IPC(IP:= DWORD#0, PORT:= WORD#0 , TIME_OUT:= timeout1, IP_C:= IP_C, S_BUF:= COM.S_BUF, R_BUF:= COM.R_BUF, TLS_CONFIG_IN := COM.TLS_CONFIG, useTls:= COM.TLS); (* MQTT Steuerkanal *)

TON_WAIT(IN:=step = last_step AND step > 0,PT:=timeout2);
last_step := step;


(* revision history


*)

END_FUNCTION_BLOCK

// MQTT/Function/InsertStringToBufferAndLength
//returnds new pos in buff
FUNCTION InsertStringToBufferAndLength : UINT
VAR_INPUT
	Str:POINTER TO STRING;
	//address to buffer
	buff:POINTER TO BYTE;
	//Start to insert
	pos:UINT;
	//size of buffer
	//size:UINT;
END_VAR
VAR
	length:UINT;
END_VAR

length := CommonTypesAndFunctions.LEN(Str);
buff[pos]:= OSCAT_BASIC.BYTE_OF_DWORD(in:= length, N:= 1);
buff[pos+1]:= OSCAT_BASIC.BYTE_OF_DWORD(in:= length, N:= 0);

MEM.MemMove(pSource:= str, pDestination:= ADR(buff[pos+2]), uiNumberOfBytes:= length);
InsertStringToBufferAndLength := pos + length + 2;

END_FUNCTION

// MQTT/Function/DoRemainingLength
FUNCTION DoRemainingLength : USINT
VAR_INPUT
	buffer:POINTER TO BYTE;
	RemainingLength:UINT;
	
END_VAR
VAR
	LocalLength:LINT;
	LocalBuffer:ARRAY[0..3]OF BYTE;
	BufferIndex:UINT := 0;
	TmpByte:BYTE;
END_VAR

//check if we have to move data for inserting remaining length
//borders are given in the mqtt doku
//
IF RemainingLength <= 128 THEN
	buffer[1] := UINT_TO_BYTE(RemainingLength);
	DoRemainingLength := 0;
ELSE
	LocalLength := RemainingLength;
	REPEAT
		TmpByte := LINT_TO_BYTE(LocalLength MOD 128);
		LocalLength := LocalLength / 128;
		IF LocalLength > 0 THEN
			TmpByte := TmpByte OR 128;
		END_IF
		LocalBuffer[BufferIndex] := TmpByte; 
		BufferIndex := BufferIndex +1;
	UNTIL 
		LocalLength <= 0 
	END_REPEAT
	//now move mem	
	//buffer index points to NEXT field, so sub 1
	MEM.MemMove(pSource:= buffer+2, pDestination:= buffer + 2 + BufferIndex - 1 , uiNumberOfBytes:= RemainingLength);
	CASE BufferIndex OF
		2: 	buffer[1]:= LocalBuffer[0];
			buffer[2]:= LocalBuffer[1];
			DoRemainingLength := 1;
		3:	buffer[1]:= LocalBuffer[0];
			buffer[2]:= LocalBuffer[1];
			buffer[3]:= LocalBuffer[2];
			DoRemainingLength := 2;
		4:	buffer[1]:= LocalBuffer[0];
			buffer[2]:= LocalBuffer[1];
			buffer[3]:= LocalBuffer[2];
			buffer[4]:= LocalBuffer[3];
			DoRemainingLength := 3;
		
	END_CASE
	
END_IF

END_FUNCTION

// MQTT/Docs/Doku
PROGRAM Doku
VAR
END_VAR

(*

Hello There,

with this library you are able to send and recvice MQTT paket on all QoS levels 0-2.

Use Pubish to publish data(Strings and binary),

Use subscribe to receive MQTT data. On Subscribe you can tell the FB if you are expecting an String as data, so you will get one on the pointer output.

How to use you can see in the example and testCase FB. This is my Test Case an it does up to 100 send and receives per second on an raspberry PI 1+ connectet to an mosquitto broker on an 
windows 10 maschine.

If you find errors, or anny instability, tell me, i will have a look.

TLS works fine without certificates.

This Projekt i using some parts of the grat OSCAT libs, so take a look at oscat.de

Greatings 

*)

END_PROGRAM

// MQTT/Function Blocks/HandleSplitTopic
FUNCTION_BLOCK HandleSplitTopic
VAR_INPUT
	
END_VAR
VAR_OUTPUT
END_VAR
VAR
		
	MySplitTopic:SPLIT_TOPIC;
	
	InitFull:BOOL;
	InitLow:BOOL;
	//this is going to be a pointer to a array of uint to store the string length(and so memmory size) in the string array 
	SplitLength:POINTER TO UINT;
	TopicsLevel:UINT;
	SplitElementSize:UINT;
	
	CountSizeExceeded:ULINT;
	TopicsIndexMax:UINT;
	dynMemUsage:POINTER TO UDINT;
	MemoryValid: BOOL;

END_VAR

{info 'TODO test of zeros in strings'}

(*use FOR high change OF topic, needs more ram, saves TIME...
allocates all memory for the string arrays and strings
usefull for often changed topics like receive publish
*)
METHOD FullInit :BOOL

VAR_INPUT
	TopicsLevelInit:UINT;
	SplitElementSizeInit:UINT;
	dynMemUsageInit:POINTER TO UDINT;
	
END_VAR
VAR
	iu:UINT;
	
END_VAR

dynMemUsage := dynMemUsageInit;
destroy();

InitFull := FALSE;
InitLow := FALSE;

TopicsLevel := TopicsLevelInit;
SplitElementSize := SplitElementSizeInit + 1;//add 1 for trailing 0
IF TopicsLevel > 0 THEN
	TopicsIndexMax := TopicsLevel - 1;
ELSE
	TopicsIndexMax := 0;
END_IF

{warning disable C0033}
//get memory for array of pointer to strings
{info 'semaphore'}
MySplitTopic.Topics := __NEW(POINTER TO STRING, TopicsLevel);
IF MySplitTopic.Topics = 0 THEN
	FullInit := FALSE;
	RETURN;		
END_IF
dynMemUsage^ := dynMemUsage^ + TopicsLevel * SIZEOF(MySplitTopic.Topics^);
FOR iu := 0 TO TopicsLevel - 1 DO
	//Get memory for strings
	{info 'semaphore'}
	MySplitTopic.Topics[iu] := __NEW(BYTE, SplitElementSize);	
	IF MySplitTopic.Topics[iu] = 0 THEN
		FullInit := FALSE;
		RETURN;		
	END_IF
	dynMemUsage^ := dynMemUsage^ + SplitElementSize;
END_FOR
{warning restore C0033}
FullInit := TRUE;
InitFull := TRUE;
MemoryValid := TRUE;
END_METHOD

(*use for low change of topic, saves mem, needs time
dynamic allocation of memory, usefull for static stopis like compare of subscription topic
*)
METHOD LowInit : bool
VAR_INPUT
	TopicsLevelInit:UINT;
	SplitElementSizeInit:UINT;
	dynMemUsageInit:POINTER TO UDINT;
END_VAR
VAR
	iu:UINT;
	
END_VAR
dynMemUsage := dynMemUsageInit;
destroy();
InitFull := FALSE;
InitLow := FALSE;

TopicsLevel := TopicsLevelInit;
SplitElementSize :=SplitElementSizeInit;
IF TopicsLevel > 0 THEN
	TopicsIndexMax := TopicsLevel - 1;
ELSE
	TopicsIndexMax := 0;
END_IF
{warning disable C0033}
//get memory for array of pointer to string 

MySplitTopic.Topics := __NEW(POINTER TO STRING, TopicsLevel);
IF MySplitTopic.Topics = 0 THEN
	LowInit := FALSE;
	RETURN;		
END_IF
{info 'semaphore'}
dynMemUsage^ := dynMemUsage^ + TopicsLevel * SIZEOF(MySplitTopic.Topics^);
//get memory for array of length of strings
{info 'semaphore'}
SplitLength := __NEW(POINTER TO STRING, TopicsLevel);
IF SplitLength = 0 THEN
	LowInit := FALSE;
	RETURN;		
END_IF

dynMemUsage^ := dynMemUsage^ + TopicsLevel * SIZEOF(SplitLength^);
{warning restore C0033}
MemoryValid := TRUE;
LowInit := TRUE;
InitLow := TRUE;
END_METHOD

METHOD destroy : bool
VAR_INPUT
END_VAR
VAR
	iu:UINT;
END_VAR
GVL_MQTT.ProgNum := PROG_NUM.DESTROY_SPLIT_TOPIC;
MemoryValid := FALSE;
IF InitFull THEN
{warning disable C0033}
	FOR iu := 0 TO TopicsLevel - 1 DO
		{info 'semaphore'}
		__DELETE(MySplitTopic.Topics[iu]);
		dynMemUsage^ := dynMemUsage^ - SplitElementSize;
	END_FOR
	{info 'semaphore'}
	__DELETE(MySplitTopic.Topics);
	dynMemUsage^ := dynMemUsage^ - (TopicsLevel * SIZEOF(MySplitTopic.Topics^));
	InitFull := FALSE;
END_IF

IF InitLow THEN
	DestroyOldSplit();
	{info 'semaphore'}
	__DELETE(MySplitTopic.Topics);
	dynMemUsage^ := dynMemUsage^ - (TopicsLevel * SIZEOF(MySplitTopic.Topics^));
	{info 'semaphore'}
	__DELETE(SplitLength);
	dynMemUsage^ := dynMemUsage^ - (TopicsLevel * SIZEOF(SplitLength^));
	InitLow:= FALSE;
END_IF
{warning restore C0033}
GVL_MQTT.ProgNum := PROG_NUM.DESTROY_SPLIT_TOPIC_DONE;
END_METHOD

METHOD GetSplitTopic : pointer to SPLIT_TOPIC
VAR_INPUT
END_VAR
GetSplitTopic := ADR(MySplitTopic);
END_METHOD

METHOD FB_Exit : BOOL 
VAR_INPUT 
 bInCopyCode : BOOL; // TRUE: the exit method is called in order to leave the instance which will be copied afterwards (online change). 
END_VAR
destroy();
END_METHOD

METHOD NewTopic : TOPIC_VALID
VAR_INPUT
	//needs to be 0 terminated!
	in:POINTER TO STRING;
	//check topic, use this for subscriptio, topics from broker should be ok...
	test: BOOL;
	//Size of String, if > 0 then use this size and don't search for 0
	SizeOfString:UINT;
	
END_VAR
VAR
	StartSub:DINT ; //in codesys for mid function first String Position is 1 !!!! devil!!!! don't use anymore, take memmove
	
	i:UINT;
	//SubCount:UINT;
	SplitChar:BYTE;
	pt:POINTER TO BYTE;
	UseSize: BOOL;

END_VAR
IF (NOT InitFull AND NOT InitLow) OR NOT MemoryValid THEN
	NewTopic := TOPIC_VALID.TOPIC_NOT_VALID;
	RETURN;
END_IF 
DestroyOldSplit();
SplitChar := CommonTypesAndFunctions.GetChar(in:= '/');
GVL_MQTT.ProgNum := PROG_NUM.GetSplitTopic;
IF SizeOfString > 0 THEN
	UseSize := TRUE;
END_IF
pt := in;
WHILE (pt[i] <> 0 AND NOT UseSize) OR (UseSize AND SizeOfString > 0) DO
	SizeOfString := SizeOfString - 1;
	IF pt[i] = SplitChar  THEN

		IF NOT PushSplitLevel(str:= ADR(in^[StartSub]), len:= i - DINT_TO_UINT(StartSub)) THEN
			CountSizeExceeded := CountSizeExceeded + 1;
			//error pushing split topic
			DestroyOldSplit();
			NewTopic := TOPIC_VALID.TOPIC_NOT_VALID;
			RETURN;
		END_IF
		StartSub := i + 1;//Start Post at next after /
	END_IF
	i := i + 1;
END_WHILE
//get last Topic...
IF NOT (i = StartSub) THEN
	
	PushSplitLevel(str:= ADR(in^[StartSub]), len:= i - DINT_TO_UINT(StartSub));

END_IF
IF pt[i - 1] = SplitChar THEN
	//got one empty level at last
	PushSplitLevel(str:= in, len:= 0);//here str doesnt need to be a valid source
END_IF
IF test THEN
	NewTopic := CheckTopicValid();
	IF NewTopic = TOPIC_VALID.TOPIC_NOT_VALID THEN
		DestroyOldSplit();
	END_IF
ELSE
	NewTopic := TOPIC_VALID.TOPIC_NO_TEST;
END_IF
END_METHOD

METHOD PushSplitLevel : bool
VAR_INPUT
	str:POINTER TO STRING;
	len:UINT;
END_VAR

VAR
	DynLength:UINT;
END_VAR
//make sure to use no more memory as allocated
IF (MySplitTopic.ValidFields >=  TopicsIndexMax) OR ((len + 1 > SplitElementSize) AND InitFull) OR NOT MemoryValid  THEN
	PushSplitLevel := FALSE;
	RETURN;
ELSE
	PushSplitLevel := TRUE;
END_IF

IF InitFull THEN
	IF len > 0 THEN
		{'info: TODO: check string length'}
		MEM.MemMove(pSource:= str, pDestination:= MySplitTopic.Topics[MySplitTopic.ValidFields], uiNumberOfBytes:= len);
	END_IF
	MySplitTopic.Topics[MySplitTopic.ValidFields]^[len] := 0;//string limiter
END_IF


IF InitLow THEN
	DynLength := len + 1;
	{warning disable C0033}
	MySplitTopic.Topics[MySplitTopic.ValidFields] := __NEW(BYTE, DynLength);
	IF MySplitTopic.Topics[MySplitTopic.ValidFields] = 0 THEN
		MemoryValid := FALSE;
		PushSplitLevel := FALSE;
		RETURN;
	END_IF
	dynMemUsage^ := dynMemUsage^ + DynLength;
	{warning restore C0033}
	IF len > 0 THEN
		MEM.MemMove(pSource:= str, pDestination:= MySplitTopic.Topics[MySplitTopic.ValidFields], uiNumberOfBytes:= len);
	END_IF
	SplitLength[MySplitTopic.ValidFields] := DynLength;
	MySplitTopic.Topics[MySplitTopic.ValidFields]^[DynLength - 1] := 0;//string limiter
END_IF

MySplitTopic.ValidFields := MySplitTopic.ValidFields + 1;
END_METHOD

METHOD DestroyOldSplit
VAR_INPUT
END_VAR
VAR
	di:DINT;
END_VAR
IF InitLow THEN
	FOR di := 0 TO MySplitTopic.ValidFields - 1 DO
{warning disable C0033}
{info 'semaphore'}
		//SysMem23.SysMemFree(dwAddress:= MySplitTopic.Topics[di], dwSize:= SplitLength[di]);
		__DELETE(MySplitTopic.Topics[di]);
		
		dynMemUsage^ := dynMemUsage^ - SplitLength[di];
{warning restore C0033}		
	END_FOR
END_IF

MySplitTopic.ValidFields := 0;
END_METHOD

//Instance needs to be subscription topic
METHOD CheckTopicMatchToMe : TOPIC_MATCH
VAR_INPUT
	//topic to compare with, here the topic from broker
	with:POINTER TO SPLIT_TOPIC;
END_VAR
VAR
	i:uINT;
	pt:POINTER TO BYTE;
	wildcard:BYTE;
END_VAR
IF NOT MemoryValid THEN
		CheckTopicMatchToMe := TOPIC_MATCH.TOPIC_NO_MEMORY;
 	RETURN;
END_IF

wildcard := CommonTypesAndFunctions.GetChar(in:= '#');
FOR i := 0 TO MIN(MySplitTopic.ValidFields - 1, with^.ValidFields - 1) DO
	pt := MySplitTopic.Topics[i]; 
	IF pt^ = wildcard THEN
		//from here its mine
		CheckTopicMatchToMe := TOPIC_MATCH.TOPIC_MATCHES;
		RETURN;
	END_IF
	IF NOT CheckTopicLevel(s1:= with^.Topics[i] , s2:= MySplitTopic.Topics[i]) THEN
		CheckTopicMatchToMe := TOPIC_MATCH.TOPIC_DONT_MATCHES;
		RETURN;
	END_IF  
END_FOR
//if here and there are further topics then its note mine
IF MySplitTopic.ValidFields = with^.ValidFields THEN
	CheckTopicMatchToMe := TOPIC_MATCH.TOPIC_MATCHES;
	RETURN;
END_IF
pt := ADR(MySplitTopic.Topics[i]);
IF MySplitTopic.ValidFields > with^.ValidFields AND 
	pt^ = wildcard THEN
	//check last Subscription topic if '#'
	CheckTopicMatchToMe := TOPIC_MATCH.TOPIC_MATCHES;
ELSE
	CheckTopicMatchToMe := TOPIC_MATCH.TOPIC_DONT_MATCHES;
END_IF
END_METHOD

METHOD CheckTopicValid : TOPIC_VALID
VAR_INPUT
END_VAR
VAR
	
	i:UINT;
	
END_VAR
IF NOT MemoryValid THEN
	RETURN;
END_IF
FOR i := 0 TO MySplitTopic.ValidFields - 1 DO
	IF (CommonTypesAndFunctions.find(STR1:= MySplitTopic.Topics[i], STR2:= ADR('#')) >= 0) AND (CommonTypesAndFunctions.len(STR:= MySplitTopic.Topics[i]) > 1) THEN
		//error # within topic
		CheckTopicValid := TOPIC_VALID.TOPIC_NOT_VALID;
		RETURN;
		
	END_IF
	IF (CommonTypesAndFunctions.find(STR1:= MySplitTopic.Topics[i], STR2:= ADR('+')) >= 0) AND (CommonTypesAndFunctions.len(STR:= MySplitTopic.Topics[i]) > 1) THEN
		//error + within topic
		CheckTopicValid := TOPIC_VALID.TOPIC_NOT_VALID;
		RETURN;
	END_IF
		IF (CommonTypesAndFunctions.find(STR1:= MySplitTopic.Topics[i], STR2:= ADR('#')) >= 0) AND (i <> MySplitTopic.ValidFields - 1) THEN
		//error # not at lowest topic
		CheckTopicValid := TOPIC_VALID.TOPIC_NOT_VALID;
		RETURN;
	END_IF
END_FOR
CheckTopicValid := TOPIC_VALID.TOPIC_VALID;
END_METHOD

END_FUNCTION_BLOCK

// MQTT/Function/CheckTopicLevel
//true if levels the same
FUNCTION CheckTopicLevel : bool
VAR_INPUT
	//String from Broker
	s1:POINTER TO STRING;
	//Subscribe String
	s2:POINTER to STRING;
END_VAR
VAR
	LenS1: UINT;
END_VAR

CheckTopicLevel := FALSE;
//test Wildcard
IF (s2^[0] = CommonTypesAndFunctions.GetChar(in:= '+')) THEN //(s2[0] = GetChar(in:= '#')) OR  don't check # here
	CheckTopicLevel := TRUE;
	RETURN;	
END_IF
LenS1 := CommonTypesAndFunctions.len(STR:= s1); 
IF (LenS1 <> CommonTypesAndFunctions.len(STR:= s2)) THEN 
	RETURN;
END_IF//if len not eval then return
IF (CommonTypesAndFunctions.find(STR1:= s1, STR2:= s2) >= 0) OR (LenS1 = 0)THEN
	CheckTopicLevel := TRUE;
END_IF

END_FUNCTION

// MQTT/Function/DoRemainingLengthBevor
//here no move of data, calc remainig length bevor moving topic and paylod, use this for 
//borders are given in the mqtt doku
//use this for publish pakets

FUNCTION DoRemainingLengthBevor : USINT
VAR_INPUT
	//points to start of buffer, not to start of remainig length!
	buffer:POINTER TO BYTE;
	SizeTopic:UDINT;
	SizePayload:UDINT;
	InQoS:QoS;
	
END_VAR
VAR
	RemainingLength:UDINT;
	LocalLength:LINT;
	LocalBuffer:ARRAY[0..3]OF BYTE;
	BufferIndex:UINT := 0;
	TmpByte:BYTE;
END_VAR


	
RemainingLength := SizeTopic + SizePayload;
	
RemainingLength := RemainingLength + 2;//add topic size encoding space
IF NOT (InQoS = QoS.AtMostOnce) THEN
	RemainingLength := RemainingLength + 2;//add space for paket identifier
END_IF

IF RemainingLength <= 128 THEN
	buffer[1] := UDINT_TO_BYTE(RemainingLength);
	DoRemainingLengthBevor := 0;
ELSE
	LocalLength := RemainingLength;
	REPEAT
		TmpByte := LINT_TO_BYTE(LocalLength MOD 128);
		LocalLength := LocalLength / 128;
		IF LocalLength > 0 THEN
			TmpByte := TmpByte OR 128;
		END_IF
		LocalBuffer[BufferIndex] := TmpByte; 
		BufferIndex := BufferIndex +1;
	UNTIL 
		LocalLength <= 0 
	END_REPEAT
	CASE BufferIndex OF
		2: 	buffer[1]:= LocalBuffer[0];
			buffer[2]:= LocalBuffer[1];
			DoRemainingLengthBevor := 1;
		3:	buffer[1]:= LocalBuffer[0];
			buffer[2]:= LocalBuffer[1];
			buffer[3]:= LocalBuffer[2];
			DoRemainingLengthBevor := 2;
		4:	buffer[1]:= LocalBuffer[0];
			buffer[2]:= LocalBuffer[1];
			buffer[3]:= LocalBuffer[2];
			buffer[4]:= LocalBuffer[3];
			DoRemainingLengthBevor := 3;
		
	END_CASE
	
END_IF

END_FUNCTION

// MQTT/Function/GetRemainingLength
FUNCTION GetRemainingLength : REMAINING_LENGTH_RETURN
VAR_INPUT
	//Pointer to Buffer
	Buff:POINTER TO BYTE;
	//Start of data in Buffer
	pos:UINT;
	//
	BuffSize:UDINT;
	//BuffSize:UINT;
END_VAR
VAR
	BufferIndex:UINT := 1;
	Multipler:UDINT := 1;
	TmpByte:BYTE;
END_VAR

GetRemainingLength.Error := FALSE;
GetRemainingLength.SizeRemainingLength:= 0;

GetRemainingLength.BuffToSmall := FALSE;
BufferIndex := pos + 1;
REPEAT
	IF BufferIndex > (BuffSize - 1) THEN
		GetRemainingLength.BuffToSmall := TRUE;
	ELSE
		TmpByte := Buff[BufferIndex];
		BufferIndex := BufferIndex + 1;
		GetRemainingLength.RemainingLength := GetRemainingLength.RemainingLength + (TmpByte AND 127) * Multipler;
		Multipler := Multipler *128;
		IF Multipler > 128*128*128 THEN
			GetRemainingLength.RemainingLength := 0;//lengt 0 if broken
			GetRemainingLength.Error := TRUE;
		END_IF
	END_IF
	GetRemainingLength.SizeRemainingLength := GetRemainingLength.SizeRemainingLength + 1;
UNTIL
	TmpByte.7 = FALSE OR GetRemainingLength.BuffToSmall
	//TmpByte.7 = FALSE  OR GetRemainingLength.RemainingLength = 0 OR GetRemainingLength.BuffToSmall
END_REPEAT
GetRemainingLength.IndexAfterRemainingLength := BufferIndex;

END_FUNCTION

// MQTT/Function Blocks/MQTTPublish
(*be aware, don't change payload and topic until send is done!!!

*)

FUNCTION_BLOCK MQTTPublish EXTENDS MQTTBase
VAR_INPUT
	(*here your topic*)
	Topic:POINTER TO STRING;
	(*here the payload String*)
	PayloadString:POINTER TO STRING;
	(*set this to true to publish a string, else the data is expected on Payload*)
	PublishAsString:BOOL;
	(*binary payload*)
	Payload:POINTER TO  BYTE;
	(*length of binary payload*)
	PayloadLength:UDINT;
	(*QoS Level*)
	QoSIn:QoS;
	//Message is retain?
	MRetain: BOOL;
	//send on positiv edge, be aware, don't change payload and topic until send is done!!!
	send: BOOL;
	

END_VAR
VAR_OUTPUT
	//sucsessfull transmittet
	done:BOOL;
	//trying to send
	sendActive: BOOL;
	//Timout of sending while connection io --> to much load
	SendTimeout: BOOL;
	//count of publish send sucsessfull
	CountSend:ULINT;

END_VAR

VAR
	requestToSend:BOOL;
	TriggerEdge:Standard.R_TRIG;
	//paket gone out
	WasSendet: BOOL;
	TimeToResponse:CAA.TICK;
	LastSend:CAA.TICK;
	MyOutData:DATA_TO_BROKER;
	//timeout timer
	SendTimeOutTime:ton;
	//Data was allready builded
	dataBuild: BOOL;
END_VAR

SUPER^();
//if not config, then leave
IF NOT DbPointerIo THEN RETURN; END_IF;
GVL_MQTT.ProgNum := PROG_NUM.Publish;
{info 'TODO check this, messeg is repeated!'}
TriggerEdge(CLK:= send AND MQTT_IN_OUT^.BROKER_CONNECTED);

IF NOT MQTT_IN_OUT^.BROKER_CONNECTED THEN
	//no connection, reset
	WasSendet := FALSE;
	MyOutData.PaketData.DUP := FALSE;
END_IF

done := FALSE;

IF TriggerEdge.Q THEN
	requestToSend := TRUE;
END_IF

IF requestToSend AND NOT dataBuild THEN
	dataBuild := TRUE;
	//build data	
	MyOutData.PaketData.MqttTopicLength := CommonTypesAndFunctions.LEN(Topic);
	//don't sent zero lengt topics...
	IF  MyOutData.PaketData.MqttTopicLength > 0 THEN
		MyOutData.PaketData.MessageType := MESSAGETYPE.PUBLISH;
		MyOutData.PaketData.MessageRetain := MRetain;
		MyOutData.PaketData.MessageQoS := QoSIn;
		IF PublishAsString THEN
			MyOutData.PaketData.MqttPayloadLength := CommonTypesAndFunctions.LEN(PayloadString);
			MyOutData.PaketData.MqttPayload := PayloadString;
		ELSE
			MyOutData.PaketData.MqttPayloadLength := PayloadLength;
			MyOutData.PaketData.MqttPayload := Payload;
		END_IF
		MyOutData.PaketData.MqttTopic := Topic;
		
		//WasSendet := TRUE;
		LastSend := TICKS.GetTick(xDummy:= TRUE);
	ELSE
		{info 'check if we want to diplay topic error'}
		;
	END_IF

END_IF

IF requestToSend AND NOT WasSendet AND MQTT_IN_OUT^.BROKER_CONNECTED THEN
	//try to publish
	IF MQTT_IN_OUT^.handleFB^.Publish(data:=ADR(MyOutData)) THEN
		WasSendet := TRUE;
	ELSE
		WasSendet := FALSE;
	END_IF
END_IF


IF MyOutData.PaketData.SendSucsess THEN //sucsses set by HANDLE_MQTT
	MyOutData.PaketData.SendSucsess := FALSE;
	//paket away...
	WasSendet := FALSE;
	requestToSend := FALSE; 
	done := TRUE;
	dataBuild := FALSE;
	MyOutData.PaketData.DUP := FALSE;
	TimeToResponse := TICKS.GetTick(xDummy:= TRUE) - LastSend;
	CountSend := CountSend + 1;
END_IF

SendTimeOutTime(IN:= requestToSend, PT:= MyConstants.SENDING_TIMEOUT);
SendTimeout := SendTimeOutTime.Q;

sendActive := requestToSend;

END_FUNCTION_BLOCK

// MQTT/Function Blocks/MQTTBase
FUNCTION_BLOCK MQTTBase
VAR_INPUT

END_VAR
	
VAR_OUTPUT
END_VAR
VAR
	MQTT_IN_OUT:POINTER TO MQTT_IN_OUT;
	//Set to true if get DB Pointer 
	DbPointerIo:BOOL;
	TokenRequested: BOOL;
	RTrig:r_trig;
	//config for boot up
	COM_CONFIG:COM_CONFIG;
END_VAR

VAR_IN_OUT
			
END_VAR

IF not DbPointerIo THEN RETURN; END_IF

METHOD SetMqttInOut : INT
VAR_INPUT
	MQTT_IN_OUT:POINTER TO MQTT_IN_OUT;
END_VAR
THIS^.MQTT_IN_OUT := MQTT_IN_OUT;
DbPointerIo := TRUE;
END_METHOD

END_FUNCTION_BLOCK

// MQTT/Function Blocks/MQTTSubscribe
(*use this to subscribe to a topic, if the topic you want to subscribe isn't valid you get an error on output SubscribeFail,

subscribing now uses callbacks for received publsih packets. you have to pass a FB instance which implements the "MQTT_SUBSCRIBE_CALLBACK" interface.
after reciving a matching topic to the subscription topic, the method PublisReceived() of the FB is called. The call passes all needed information to the callback.
in the called method you can differ the topic or payload more finer if needed. See the ListAllValueCallback() and ListStringCallback for example.
they using a list to the exact topic. So you can subscribe to a topic with wildcard or fix topic with coded payload, and the list FBs doing the fine stuff.
 *)
FUNCTION_BLOCK MQTTSubscribe EXTENDS MQTTBase
VAR_INPUT
	(*set to true to subscribe, set to false to unsubscribe*)
	Subscribe:BOOL;
	(*your topic string*)
	Topic:POINTER TO STRING;
	(*QoS level*)
	QoSSubscribe:QoS;
	(*set to true is you want an string as output, if so you get the String on PayloadString, else
		you get binary data on payload*)
	ExpectingString:BOOL;
	//callback FB
	Callback:MQTT_SUBSCRIBE_CALLBACK;
END_VAR
VAR_OUTPUT
	SubscribeDone: BOOL;
	//Timout of sending(subscribe paket) while connection io --> to much load
	SendTimeout: BOOL;
	(*error if subscribtion on broker fails or if topic isn't valid*)
	SubscribeFail: BOOL;
	(*here you get your topic check*)
	TopicValid:TOPIC_VALID;
	
END_VAR
VAR
	
	SubscribeRising:R_TRIG;
	SubscribeFalling:F_TRIG;
	NeedSubscribe: BOOL;
	NeedUnsubscribe: BOOL;
	
	SubscribeWasSended: BOOL;
	UnsubscribeWasSended: BOOL;
	MyOutData:DATA_TO_BROKER;
	TimeToResponse:CAA.TICK;
	LastSend:CAA.TICK;
	SendTimeOutTime:ton;
	ReceivedQoS:QoS;
	MySplitTopic:HandleSplitTopic;
	//received publishs
	ReceivedPublishs:ULINT;
	
	init:BOOL:=FALSE;
	iu:UINT;
END_VAR

SUPER^();
//if not config, then leave
IF NOT DbPointerIo THEN RETURN; END_IF;
GVL_MQTT.ProgNum := PROG_NUM.Subscribe;
SubscribeFalling(CLK:= Subscribe);
SubscribeRising(CLK:= Subscribe);

IF NOT init THEN
	COM_CONFIG := MQTT_IN_OUT^.COM_CONFIG;
	MySplitTopic.LowInit(TopicsLevelInit:= COM_CONFIG.MaxTopicLevels, SplitElementSizeInit:= COM_CONFIG.MaxTopicElementSize, dynMemUsageInit:= ADR(MQTT_IN_OUT^.dynMemUsage));
	init:= TRUE;
END_IF

IF NOT MQTT_IN_OUT^.BROKER_CONNECTED AND Subscribe THEN
	//reconnect after disconnect
	NeedSubscribe := TRUE;
	SubscribeDone := FALSE;
	SubscribeWasSended := FALSE;
	UnsubscribeWasSended := FALSE;
END_IF

IF SubscribeRising.Q THEN
	NeedSubscribe := TRUE;
END_IF


IF SubscribeFalling.Q THEN
	NeedUnsubscribe := TRUE;
END_IF


{info 'reconnect or wait or or or or ....'}
//have to unsubscribe if callback wasn't registered
IF MyOutData.PaketData.CallbackError THEN
	NeedUnsubscribe := TRUE;
	SubscribeFail := TRUE;
END_IF

IF NeedSubscribe AND NOT SubscribeWasSended AND MQTT_IN_OUT^.InFree AND MQTT_IN_OUT^.BROKER_CONNECTED THEN
 
	TopicValid := MySplitTopic.NewTopic(in:= Topic, test:= TRUE, SizeOfString:= 0);  
	IF TopicValid = TOPIC_VALID.TOPIC_VALID THEN
		//try to subscribe
		SubscribeWasSended := TRUE;
		//send free
		MQTT_IN_OUT^.IN := ADR(MyOutData);
		MQTT_IN_OUT^.InFree := FALSE;
		MyOutData.PaketData.MessageType := MESSAGETYPE.SUBSCRIBE;
		MyOutData.PaketData.MessageQoS := QoSSubscribe;
		MyOutData.PaketData.Callback := Callback;
		MyOutData.PaketData.MqttTopic := Topic;
		MyOutData.PaketData.MqttTopicLength := CommonTypesAndFunctions.LEN(Topic);
		MyOutData.PaketData.SplitTopic := ADR(MySplitTopic);
		MyOutData.PaketData.ExpectingString := ExpectingString;
	
		SubscribeFail := FALSE;
	ELSE
		NeedSubscribe := FALSE;
		SubscribeFail := TRUE;
	END_IF
	//ReleaseToken();
END_IF

IF NeedUnsubscribe AND NOT UnsubscribeWasSended AND MQTT_IN_OUT^.InFree AND MQTT_IN_OUT^.BROKER_CONNECTED THEN
	//try to unsubscribe
	UnsubscribeWasSended := TRUE;
	//send free
	MQTT_IN_OUT^.IN := ADR(MyOutData);
	MQTT_IN_OUT^.InFree := FALSE;
	MyOutData.PaketData.Callback := Callback;
	MyOutData.PaketData.MessageType := MESSAGETYPE.UNSUBSCRIBE;
	MyOutData.PaketData.MqttTopic := Topic;
	MyOutData.PaketData.MqttTopicLength := CommonTypesAndFunctions.LEN(Topic);
	//ReleaseToken();
END_IF

//place behinde send, so leave "Token" to rest....
//here for Subscribe
IF MyOutData.PaketData.SendSucsess AND MyOutData.PaketData.MessageType = MESSAGETYPE.SUBSCRIBE THEN //scusses set by HANDLE_MQTT
	MyOutData.PaketData.SendSucsess := FALSE;
	//paket away...
	SubscribeWasSended := FALSE;
	NeedSubscribe := FALSE; 
	SubscribeDone := TRUE;
	TimeToResponse := TICKS.GetTick(xDummy:= TRUE) - LastSend;
	ReceivedQoS := MyOutData.PaketData.SubackQoS;
	IF ReceivedQoS = QoS.Fail THEN
		SubscribeFail := TRUE;
	ELSE
		SubscribeFail := FALSE;	
	END_IF
	
END_IF

//here for Unubscribe
IF MyOutData.PaketData.SendSucsess AND MyOutData.PaketData.MessageType = MESSAGETYPE.UNSUBSCRIBE THEN //scusses set by HANDLE_MQTT
	MyOutData.PaketData.SendSucsess := FALSE;
	//paket away...
	UnsubscribeWasSended := FALSE;
	NeedUnsubscribe := FALSE; 
	SubscribeDone := FALSE;
	TimeToResponse := TICKS.GetTick(xDummy:= TRUE) - LastSend;
END_IF

SendTimeOutTime(IN:= NeedSubscribe OR NeedUnsubscribe, PT:= MyConstants.SENDING_TIMEOUT);
SendTimeout := SendTimeOutTime.Q;

END_FUNCTION_BLOCK

// MQTT/Interfaces/MQTT_SUBSCRIBE_CALLBACK
(*this is the interface for subscription callbacks.
you can implement it in you one FBs and pass this to the CallbackStock or subscription FB*)
INTERFACE MQTT_SUBSCRIBE_CALLBACK

METHOD PublishReceived : bool
VAR_INPUT
	//Collection of received Data
	Data:CALLBACK_DATA;
END_VAR
END_METHOD

END_INTERFACE

// MQTT/Function Blocks/CallbackFBs/ListCallbacks/ListStringCallback
FUNCTION_BLOCK ListStringCallback IMPLEMENTS MQTT_SUBSCRIBE_CALLBACK
VAR_INPUT
END_VAR
VAR_OUTPUT
END_VAR
VAR
	MyListData:POINTER TO LIST_STRING_CALLBACK_DATA;
	MyLengthOfData:ULINT;
	ListSplitTopic:BOOL;
	ListSplitPayload:BOOL;
	SplitCharPayload:BYTE;
	

END_VAR

METHOD PublishReceived : BOOL
VAR_INPUT
	//Collection of received Data
	Data:CALLBACK_DATA;

END_VAR
VAR
	i:ULINT;
	StrPt:POINTER TO STRING(255);
	SplitPos:DINT;
END_VAR
//now search the right topic 
IF ListSplitTopic THEN
	FOR i := 0 TO MyLengthOfData - 1 DO
		IF CommonTypesAndFunctions.StrEquals(str1:= Data.TopicOutSplit^.Topics[Data.TopicOutSplit^.ValidFields - 1], str2:= MyListData[i].SubTopic) THEN
			//MyListData[i].Target^ := Data.PayloadString^;
			MEM.MemMove(pSource:= Data.PayloadString, pDestination:= MyListData[i].Target, uiNumberOfBytes:= TO_UINT(data.PayloadSize + 1));
			PublishReceived := TRUE;
		END_IF
	END_FOR
END_IF

IF ListSplitPayload THEN
	FOR i := 0 TO MyLengthOfData - 1 DO
		IF CommonTypesAndFunctions.StrEqualsAtStartWithDelimiter(str1:= MyListData[i].SubTopic, str2:= Data.PayloadString, delimiter:= SplitCharPayload) THEN
			//now search split char
			StrPt := Data.PayloadString;
			SplitPos := CommonTypesAndFunctions.find(str1 := StrPt, str2:= ADR(SplitCharPayload));
			StrPt := StrPt + TO_DWORD(SplitPos) + 1;
			//MyListData[i].Target^ := StrPt^;
			MEM.MemMove(pSource:= Data.PayloadString, pDestination:= MyListData[i].Target, uiNumberOfBytes:= TO_UINT(data.PayloadSize + 1 - TO_UDINT(SplitPos)) );
			PublishReceived := TRUE;
		END_IF
	END_FOR
	
END_IF
END_METHOD

//ints FB to split packets at lowest payload level
METHOD InitAsSplitTopic : BOOL
VAR_INPUT
	ListData:POINTER TO LIST_STRING_CALLBACK_DATA;
	//Count of List Data
	LengthOfData:ULINT;

END_VAR
MyListData :=ListData;
MyLengthOfData := LengthOfData;
ListSplitTopic := TRUE;
ListSplitPayload := FALSE;
END_METHOD

(*inits FB, callback methoth then checks if the payload ist the same in the first characters as in the template
make sure to receive a string payload!
*)
METHOD InitAsSplitPayload : BOOL
VAR_INPUT
	ListData:POINTER TO LIST_STRING_CALLBACK_DATA;
	//Count of List Data
	LengthOfData:ULINT;
	//spliting character
	SplitChar:BYTE;
END_VAR
MyListData :=ListData;
MyLengthOfData := LengthOfData;
ListSplitTopic := FALSE;
ListSplitPayload := TRUE;
SplitCharPayload := SplitChar;
END_METHOD

END_FUNCTION_BLOCK

// MQTT/TestCases/TestcaseCheckTopivValid
FUNCTION_BLOCK TestcaseCheckTopivValid
VAR_INPUT
END_VAR
VAR_OUTPUT
END_VAR
VAR

	
	
	t1:HandleSplitTopic;
	s100:STRING[101]:='1111111111111111111111111111111111111111111111111111111111111111111111111111111111111111111111111111';
	splus:STRING:='+';
	ssharp:STRING:='#';
	stest:STRING:='test';
	valids:ARRAY[0..30]OF STRING :=['/+//sdf/test1',
									'/sd//',
									'test1/+/rest/#',
									'test1/#',
									'test1/topic2/+/Topic3/+/5636/ggesd',
									'///',
									'///+//sdf/test1//',
									'//+//sdf/test1/',
									'#',
									'',
									'',
									'',
									'',
									'',
									''];
	falses:ARRAY[0..30]OF STRING :=['test1/topic2/+/Topic3#/',
									'test1/#/topic2/+/Topic3/#456',
									'test1+',
									'test1/#/topic2/+/Topic3/+/5636/ggesd',
									'test1#',
									'',
									'',
									'',
									'',
									'',
									'',
									'',
									'',
									'',
									''];
	s1:STRING(64000);
	valid:TOPIC_VALID;
	pts:ARRAY[0..20] OF POINTER TO STRING; 
	sp:POINTER TO SPLIT_TOPIC;
	COM_CONFIG: COM_CONFIG;
	dynMemUsage: UDINT;
END_VAR

	(*GetSplitTopic(in:= 'test1/topic2/+/Topic3#/', Target:= ADR(dis1), CountSplitTopicSizeExceeded:= ADR(CountSplitTopicSizeExceeded));
	
	GetSplitTopic(in:= 'test1/#/topic2/+/Topic3/#456', Target:= ADR(dis2), CountSplitTopicSizeExceeded:= ADR(CountSplitTopicSizeExceeded));
	GetSplitTopic(in:= 'test1/+/rest/#', Target:= ADR(dis3), CountSplitTopicSizeExceeded:= ADR(CountSplitTopicSizeExceeded));
	GetSplitTopic(in:= 'test1/#', Target:= ADR(dis4), CountSplitTopicSizeExceeded:= ADR(CountSplitTopicSizeExceeded));
	GetSplitTopic(in:= 'test1/topic2/+/Topic3/+/5636/ggesd', Target:= ADR(dis5), CountSplitTopicSizeExceeded:= ADR(CountSplitTopicSizeExceeded));
	GetSplitTopic(in:= 'test1/#/topic2/+/Topic3/+/5636/ggesd', Target:= ADR(dis6), CountSplitTopicSizeExceeded:= ADR(CountSplitTopicSizeExceeded));
	GetSplitTopic(in:= 'test1#', Target:= ADR(dis7), CountSplitTopicSizeExceeded:= ADR(CountSplitTopicSizeExceeded));
	GetSplitTopic(in:= 'test1+', Target:= ADR(dis8), CountSplitTopicSizeExceeded:= ADR(CountSplitTopicSizeExceeded));
	GetSplitTopic(in:= '/+//sdf/test1', Target:= ADR(dis9), CountSplitTopicSizeExceeded:= ADR(CountSplitTopicSizeExceeded));
	GetSplitTopic(in:= '//+//sdf/test1/', Target:= ADR(dis10), CountSplitTopicSizeExceeded:= ADR(CountSplitTopicSizeExceeded));
	GetSplitTopic(in:= '///+//sdf/test1//', Target:= ADR(dis11), CountSplitTopicSizeExceeded:= ADR(CountSplitTopicSizeExceeded));
	GetSplitTopic(in:= '///', Target:= ADR(dis12), CountSplitTopicSizeExceeded:= ADR(CountSplitTopicSizeExceeded));
	GetSplitTopic(in:= '/sd//', Target:= ADR(dis13), CountSplitTopicSizeExceeded:= ADR(CountSplitTopicSizeExceeded));
	Valid1:=CheckTopicValid(Target:= ADR(dis1));
	Valid2:=CheckTopicValid(Target:= ADR(dis2));
	Valid3:=CheckTopicValid(Target:= ADR(dis3));
	Valid4:=CheckTopicValid(Target:= ADR(dis4));
	Valid5:=CheckTopicValid(Target:= ADR(dis5));
	Valid6:=CheckTopicValid(Target:= ADR(dis6));
	Valid7:=CheckTopicValid(Target:= ADR(dis7));
	Valid8:=CheckTopicValid(Target:= ADR(dis8));
	Valid9:=CheckTopicValid(Target:= ADR(dis9));
	*)
	
	t1.LowInit(SplitElementSizeInit:=400, TopicsLevelInit:= 40, dynMemUsageInit:= ADR(dynMemUsage));
	valid := t1.NewTopic(in := ADR(valids[0]), test:= TRUE, SizeOfString:= 0);
	sp := t1.GetSplitTopic();
	pts[0] := sp^.Topics[0];
	pts[1] := sp^.Topics[1];
	pts[2] := sp^.Topics[2];
	pts[3] := sp^.Topics[3];
	pts[4] := sp^.Topics[4];
	pts[5] := sp^.Topics[5];
	pts[6] := sp^.Topics[6];
	pts[7] := sp^.Topics[7];
	pts[8] := sp^.Topics[8];
	valid := t1.NewTopic(in := ADR(valids[1]), test:= TRUE, SizeOfString:= 0);
	valid := t1.NewTopic(in := ADR(valids[2]), test:= TRUE, SizeOfString:= 0);
	valid := t1.NewTopic(in := ADR(valids[3]), test:= TRUE, SizeOfString:= 0);
	valid := t1.NewTopic(in := ADR(valids[4]), test:= TRUE, SizeOfString:= 0);
	valid := t1.NewTopic(in := ADR(valids[5]), test:= TRUE, SizeOfString:= 0);
	valid := t1.NewTopic(in := ADR(valids[6]), test:= TRUE, SizeOfString:= 0);
	valid := t1.NewTopic(in := ADR(valids[7]), test:= TRUE, SizeOfString:= 0);
	valid := t1.NewTopic(in := ADR(valids[8]), test:= TRUE, SizeOfString:= 0);
	
	valid := t1.NewTopic(in := ADR(falses[0]), test:= TRUE, SizeOfString:= 0);
	valid := t1.NewTopic(in := ADR(falses[1]), test:= TRUE, SizeOfString:= 0);
	valid := t1.NewTopic(in := ADR(falses[2]), test:= TRUE, SizeOfString:= 0);
	valid := t1.NewTopic(in := ADR(falses[3]), test:= TRUE, SizeOfString:= 0);
	valid := t1.NewTopic(in := ADR(falses[4]), test:= TRUE, SizeOfString:= 0);
	valid := t1.NewTopic(in := ADR(falses[5]), test:= TRUE, SizeOfString:= 0);
	valid := t1.NewTopic(in := ADR(falses[6]), test:= TRUE, SizeOfString:= 0);
	valid := t1.NewTopic(in := ADR(falses[7]), test:= TRUE, SizeOfString:= 0);
	
	
	//now bulid some realy big topics and thest them....
	s1 :='';
	CommonTypesAndFunctions.concat(s1:= ADR(s1), s2:= ADR('/'));
	CommonTypesAndFunctions.concat(s1:= ADR(s1), s2:= ADR(s100));
	CommonTypesAndFunctions.concat(s1:= ADR(s1), s2:= ADR('/'));
	CommonTypesAndFunctions.concat(s1:= ADR(s1), s2:= ADR(splus));
	CommonTypesAndFunctions.concat(s1:= ADR(s1), s2:= ADR('/'));
	CommonTypesAndFunctions.concat(s1:= ADR(s1), s2:= ADR(s100));
	CommonTypesAndFunctions.concat(s1:= ADR(s1), s2:= ADR('/'));
	CommonTypesAndFunctions.concat(s1:= ADR(s1), s2:= ADR(s100));
	CommonTypesAndFunctions.concat(s1:= ADR(s1), s2:= ADR('/'));
	CommonTypesAndFunctions.concat(s1:= ADR(s1), s2:= ADR(ssharp));
	//valid
	valid := t1.NewTopic(in := ADR(s1), test:= TRUE, SizeOfString:= 0);
	s1 :='';
	CommonTypesAndFunctions.concat(s1:= ADR(s1), s2:= ADR('/'));
	CommonTypesAndFunctions.concat(s1:= ADR(s1), s2:= ADR(s100));
	CommonTypesAndFunctions.concat(s1:= ADR(s1), s2:= ADR('/'));
	CommonTypesAndFunctions.concat(s1:= ADR(s1), s2:= ADR(splus));
	CommonTypesAndFunctions.concat(s1:= ADR(s1), s2:= ADR('/'));
	CommonTypesAndFunctions.concat(s1:= ADR(s1), s2:= ADR(s100));
	CommonTypesAndFunctions.concat(s1:= ADR(s1), s2:= ADR('/'));
	CommonTypesAndFunctions.concat(s1:= ADR(s1), s2:= ADR(s100));
	CommonTypesAndFunctions.concat(s1:= ADR(s1), s2:= ADR('/'));
	CommonTypesAndFunctions.concat(s1:= ADR(s1), s2:= ADR(ssharp));
	CommonTypesAndFunctions.concat(s1:= ADR(s1), s2:= ADR('/'));
	//not valid # not at last pos
	valid := t1.NewTopic(in := ADR(s1), test:= TRUE, SizeOfString:= 0);
	s1 :='';
	CommonTypesAndFunctions.concat(s1:= ADR(s1), s2:= ADR('/'));
	CommonTypesAndFunctions.concat(s1:= ADR(s1), s2:= ADR(s100));
	CommonTypesAndFunctions.concat(s1:= ADR(s1), s2:= ADR('/'));
	CommonTypesAndFunctions.concat(s1:= ADR(s1), s2:= ADR(splus));
	CommonTypesAndFunctions.concat(s1:= ADR(s1), s2:= ADR('/'));
	CommonTypesAndFunctions.concat(s1:= ADR(s1), s2:= ADR(s100));
	CommonTypesAndFunctions.concat(s1:= ADR(s1), s2:= ADR(splus));
	CommonTypesAndFunctions.concat(s1:= ADR(s1), s2:= ADR('/'));
	CommonTypesAndFunctions.concat(s1:= ADR(s1), s2:= ADR(s100));
	CommonTypesAndFunctions.concat(s1:= ADR(s1), s2:= ADR('/'));
	CommonTypesAndFunctions.concat(s1:= ADR(s1), s2:= ADR(ssharp));
	
	//not valid + within topic
	valid := t1.NewTopic(in := ADR(s1), test:= TRUE, SizeOfString:= 0);
	
	s1 :='';
	CommonTypesAndFunctions.concat(s1:= ADR(s1), s2:= ADR('/'));
	CommonTypesAndFunctions.concat(s1:= ADR(s1), s2:= ADR(s100));
	CommonTypesAndFunctions.concat(s1:= ADR(s1), s2:= ADR('/'));
	CommonTypesAndFunctions.concat(s1:= ADR(s1), s2:= ADR(splus));
	CommonTypesAndFunctions.concat(s1:= ADR(s1), s2:= ADR('/'));
	CommonTypesAndFunctions.concat(s1:= ADR(s1), s2:= ADR(s100));
	CommonTypesAndFunctions.concat(s1:= ADR(s1), s2:= ADR(ssharp));
	CommonTypesAndFunctions.concat(s1:= ADR(s1), s2:= ADR('/'));
	CommonTypesAndFunctions.concat(s1:= ADR(s1), s2:= ADR(s100));
	CommonTypesAndFunctions.concat(s1:= ADR(s1), s2:= ADR('/'));
	CommonTypesAndFunctions.concat(s1:= ADR(s1), s2:= ADR(ssharp));
	
	//not valid # within topic
	valid := t1.NewTopic(in := ADR(s1), test:= TRUE, SizeOfString:= 0);

END_FUNCTION_BLOCK

// MQTT/TestCases/TestSubscribeOld
FUNCTION_BLOCK TestSubscribeOld
VAR_INPUT
END_VAR
VAR_OUTPUT
END_VAR
VAR
	MQTT_IN_OUT:MQTT_IN_OUT;
	subscribe:ARRAY[0..20] OF MQTTSubscribe;
	init: BOOL;
	i:INT;
	received:ARRAY[0..20]OF BOOL;
	CountSplitTopicSizeExceeded:ULINT;
END_VAR

IF NOT init THEN
	init := TRUE;
	FOR i := 0 TO 20 DO
		subscribe[i].SetMqttInOut(MQTT_IN_OUT := ADR(MQTT_IN_OUT));
	END_FOR
END_IF

MQTT_IN_OUT.InFree := TRUE;
(*
MQTT_IN_OUT.OUT.MqttTopic := 'r//test';
//GetSplitTopic(in:= MQTT_IN_OUT.OUT.MqttTopic, Target:= ADR(MQTT_IN_OUT.OUT.Topics), CountSplitTopicSizeExceeded:= ADR(CountSplitTopicSizeExceeded));
i:=0;
subscribe[i](
	Subscribe:= TRUE, 
	Topic:= '+//test', 
	QoSSubscribe:= 0, 
	Payload=> , 
	TopicOut=> , 
	SendTimeout=> , 
	SubscribeFail=> , 
	TopicValid=> , 
	Received=> received[i]);
MQTT_IN_OUT.OUT.MqttTopic := '/rest/zt';
//GetSplitTopic(in:= MQTT_IN_OUT.OUT.MqttTopic, Target:= ADR(MQTT_IN_OUT.OUT.Topics), CountSplitTopicSizeExceeded:= ADR(CountSplitTopicSizeExceeded));
i:=i+1;
subscribe[i](
	Subscribe:= TRUE, 
	Topic:= '#', 
	QoSSubscribe:= 0, 
	Payload=> , 
	TopicOut=> , 
	SendTimeout=> , 
	SubscribeFail=> , 
	TopicValid=> , 
	Received=> received[i]);
MQTT_IN_OUT.OUT.MqttTopic := '566//test/3565/356';
//GetSplitTopic(in:= MQTT_IN_OUT.OUT.MqttTopic, Target:= ADR(MQTT_IN_OUT.OUT.Topics), CountSplitTopicSizeExceeded:= ADR(CountSplitTopicSizeExceeded));
i:=i+1;
subscribe[i](
	Subscribe:= TRUE, 
	Topic:= '+//test/#', 
	QoSSubscribe:= 0, 
	Payload=> , 
	TopicOut=> , 
	SendTimeout=> , 
	SubscribeFail=> , 
	TopicValid=> , 
	Received=> received[i]);
MQTT_IN_OUT.OUT.MqttTopic := 'test';
//GetSplitTopic(in:= MQTT_IN_OUT.OUT.MqttTopic, Target:= ADR(MQTT_IN_OUT.OUT.Topics), CountSplitTopicSizeExceeded:= ADR(CountSplitTopicSizeExceeded));
i:=i+1;
subscribe[i](
	Subscribe:= TRUE, 
	Topic:= 'test', 
	QoSSubscribe:= 0, 
	Payload=> , 
	TopicOut=> , 
	SendTimeout=> , 
	SubscribeFail=> , 
	TopicValid=> , 
	Received=> received[i]);
MQTT_IN_OUT.OUT.MqttTopic := '/test/';
//GetSplitTopic(in:= MQTT_IN_OUT.OUT.MqttTopic, Target:= ADR(MQTT_IN_OUT.OUT.Topics), CountSplitTopicSizeExceeded:= ADR(CountSplitTopicSizeExceeded));
i:=i+1;
subscribe[i](
	Subscribe:= TRUE, 
	Topic:= 'test/', 
	QoSSubscribe:= 0, 
	Payload=> , 
	TopicOut=> , 
	SendTimeout=> , 
	SubscribeFail=> , 
	TopicValid=> , 
	Received=> received[i]);
MQTT_IN_OUT.OUT.MqttTopic := 'test/test1';
//GetSplitTopic(in:= MQTT_IN_OUT.OUT.MqttTopic, Target:= ADR(MQTT_IN_OUT.OUT.Topics), CountSplitTopicSizeExceeded:= ADR(CountSplitTopicSizeExceeded));
i:=i+1;
subscribe[i](
	Subscribe:= TRUE, 
	Topic:= 'test/test1', 
	QoSSubscribe:= 0, 
	Payload=> , 
	TopicOut=> , 
	SendTimeout=> , 
	SubscribeFail=> , 
	TopicValid=> , 
	Received=> received[i]);
MQTT_IN_OUT.OUT.MqttTopic := 'a/ret/test';
//GetSplitTopic(in:= MQTT_IN_OUT.OUT.MqttTopic, Target:= ADR(MQTT_IN_OUT.OUT.Topics), CountSplitTopicSizeExceeded:= ADR(CountSplitTopicSizeExceeded));
i:=i+1;
subscribe[i](
	Subscribe:= TRUE, 
	Topic:= 'a/+/test', 
	QoSSubscribe:= 0, 
	Payload=> , 
	TopicOut=> , 
	SendTimeout=> , 
	SubscribeFail=> , 
	TopicValid=> , 
	Received=> received[i]);
MQTT_IN_OUT.OUT.MqttTopic := '/test/etwetre/';
//GetSplitTopic(in:= MQTT_IN_OUT.OUT.MqttTopic, Target:= ADR(MQTT_IN_OUT.OUT.Topics), CountSplitTopicSizeExceeded:= ADR(CountSplitTopicSizeExceeded));
i:=i+1;
subscribe[i](
	Subscribe:= TRUE, 
	Topic:= '/test/+',//no match !!!!!
	QoSSubscribe:= 0, 
	Payload=> , 
	TopicOut=> , 
	SendTimeout=> , 
	SubscribeFail=> , 
	TopicValid=> , 
	Received=> received[i]);
MQTT_IN_OUT.OUT.MqttTopic := '/test/etwetre';
//GetSplitTopic(in:= MQTT_IN_OUT.OUT.MqttTopic, Target:= ADR(MQTT_IN_OUT.OUT.Topics), CountSplitTopicSizeExceeded:= ADR(CountSplitTopicSizeExceeded));
i:=i+1;
subscribe[i](
	Subscribe:= TRUE, 
	Topic:= '/test/+',//match !!!!!!
	QoSSubscribe:= 0, 
	Payload=> , 
	TopicOut=> , 
	SendTimeout=> , 
	SubscribeFail=> , 
	TopicValid=> , 
	Received=> received[i]);
MQTT_IN_OUT.OUT.MqttTopic := '/finance';
//GetSplitTopic(in:= MQTT_IN_OUT.OUT.MqttTopic, Target:= ADR(MQTT_IN_OUT.OUT.Topics), CountSplitTopicSizeExceeded:= ADR(CountSplitTopicSizeExceeded));
i:=i+1;
subscribe[i](
	Subscribe:= TRUE, 
	Topic:= '+/+', //match
	QoSSubscribe:= 0, 
	Payload=> , 
	TopicOut=> , 
	SendTimeout=> , 
	SubscribeFail=> , 
	TopicValid=> , 
	Received=> received[i]);
MQTT_IN_OUT.OUT.MqttTopic := '/finance';
//GetSplitTopic(in:= MQTT_IN_OUT.OUT.MqttTopic, Target:= ADR(MQTT_IN_OUT.OUT.Topics), CountSplitTopicSizeExceeded:= ADR(CountSplitTopicSizeExceeded));
i:=i+1;
subscribe[i](
	Subscribe:= TRUE, 
	Topic:= '/+', //match
	QoSSubscribe:= 0, 
	Payload=> , 
	TopicOut=> , 
	SendTimeout=> , 
	SubscribeFail=> , 
	TopicValid=> , 
	Received=> received[i]);
MQTT_IN_OUT.OUT.MqttTopic := '/finance';
//GetSplitTopic(in:= MQTT_IN_OUT.OUT.MqttTopic, Target:= ADR(MQTT_IN_OUT.OUT.Topics), CountSplitTopicSizeExceeded:= ADR(CountSplitTopicSizeExceeded));
i:=i+1;
subscribe[i](
	Subscribe:= TRUE, 
	Topic:= '+',//no match 
	QoSSubscribe:= 0, 
	Payload=> , 
	TopicOut=> , 
	SendTimeout=> , 
	SubscribeFail=> , 
	TopicValid=> , 
	Received=> received[i]);
MQTT_IN_OUT.OUT.MqttTopic := 'finance/test';
//GetSplitTopic(in:= MQTT_IN_OUT.OUT.MqttTopic, Target:= ADR(MQTT_IN_OUT.OUT.Topics), CountSplitTopicSizeExceeded:= ADR(CountSplitTopicSizeExceeded));
i:=i+1;
subscribe[i](
	Subscribe:= TRUE, 
	Topic:= 'finance/test/',//** 
	QoSSubscribe:= 0, 
	Payload=> , 
	TopicOut=> , 
	SendTimeout=> , 
	SubscribeFail=> , 
	TopicValid=> , 
	Received=> received[i]);
MQTT_IN_OUT.OUT.MqttTopic := 'finance/test';
//GetSplitTopic(in:= MQTT_IN_OUT.OUT.MqttTopic, Target:= ADR(MQTT_IN_OUT.OUT.Topics), CountSplitTopicSizeExceeded:= ADR(CountSplitTopicSizeExceeded));
i:=i+1;
subscribe[i](
	Subscribe:= TRUE, 
	Topic:= 'finance/test',//?? 
	QoSSubscribe:= 0, 
	Payload=> , 
	TopicOut=> , 
	SendTimeout=> , 
	SubscribeFail=> , 
	TopicValid=> , 
	Received=> received[i]);
MQTT_IN_OUT.OUT.MqttTopic := 'finance/test';
//GetSplitTopic(in:= MQTT_IN_OUT.OUT.MqttTopic, Target:= ADR(MQTT_IN_OUT.OUT.Topics), CountSplitTopicSizeExceeded:= ADR(CountSplitTopicSizeExceeded));
i:=i+1;
subscribe[i](
	Subscribe:= TRUE, 
	Topic:= 'finance/test/+',//?? 
	QoSSubscribe:= 0, 
	Payload=> , 
	TopicOut=> , 
	SendTimeout=> , 
	SubscribeFail=> , 
	TopicValid=> , 
	Received=> received[i]);

MQTT_IN_OUT.OUT.MqttTopic := 'finance';
//GetSplitTopic(in:= MQTT_IN_OUT.OUT.MqttTopic, Target:= ADR(MQTT_IN_OUT.OUT.Topics), CountSplitTopicSizeExceeded:= ADR(CountSplitTopicSizeExceeded));
i:=i+1;
subscribe[i](
	Subscribe:= TRUE, 
	Topic:= 'finance/#',//?match
	QoSSubscribe:= 0, 
	Payload=> , 
	TopicOut=> , 
	SendTimeout=> , 
	SubscribeFail=> , 
	TopicValid=> , 
	Received=> received[i]);
MQTT_IN_OUT.OUT.MqttTopic := 'finance/';
//GetSplitTopic(in:= MQTT_IN_OUT.OUT.MqttTopic, Target:= ADR(MQTT_IN_OUT.OUT.Topics), CountSplitTopicSizeExceeded:= ADR(CountSplitTopicSizeExceeded));
i:=i+1;
subscribe[i](
	Subscribe:= TRUE, 
	Topic:= 'finance/#',// match 
	QoSSubscribe:= 0, 
	Payload=> , 
	TopicOut=> , 
	SendTimeout=> , 
	SubscribeFail=> , 
	TopicValid=> , 
	Received=> received[i]);
MQTT_IN_OUT.OUT.MqttTopic := 'test/ff';
//GetSplitTopic(in:= MQTT_IN_OUT.OUT.MqttTopic, Target:= ADR(MQTT_IN_OUT.OUT.Topics), CountSplitTopicSizeExceeded:= ADR(CountSplitTopicSizeExceeded));
i:=i+1;
subscribe[i](
	Subscribe:= TRUE, 
	Topic:= 'test/ff/+',//no match 
	QoSSubscribe:= 0, 
	Payload=> , 
	TopicOut=> , 
	SendTimeout=> , 
	SubscribeFail=> , 
	TopicValid=> , 
	Received=> received[i]);
MQTT_IN_OUT.OUT.MqttTopic := 'test/ff';
//GetSplitTopic(in:= MQTT_IN_OUT.OUT.MqttTopic, Target:= ADR(MQTT_IN_OUT.OUT.Topics), CountSplitTopicSizeExceeded:= ADR(CountSplitTopicSizeExceeded));
i:=i+1;
subscribe[i](
	Subscribe:= TRUE, 
	Topic:= 'test/ff/#',//match 
	QoSSubscribe:= 0, 
	Payload=> , 
	TopicOut=> , 
	SendTimeout=> , 
	SubscribeFail=> , 
	TopicValid=> , 
	Received=> received[i]);
*)

END_FUNCTION_BLOCK

// MQTT/TestCases/TestMqtt
FUNCTION_BLOCK TestMqtt
VAR_INPUT
	clientID:string:='testCodesys';
END_VAR
VAR_OUTPUT
END_VAR
VAR
	MQTT:HANDLE_MQTT;
	
	MQTT_IN_OUT:MQTT_IN_OUT;
	ERROR_C:DWORD;
	ERROR_T:BYTE;
	//testPiublish: SD_MQTT.MQTTPublish;
	testPublish: ARRAY[0..100] OF MQTTPublish;
	init:BOOL := FALSE;
	sendTest: BOOL;
	testBigPublish: BOOL;
	testBigPayload: BOOL;
	testTimeBigPublish:ton;
	testTimeBigPayload:ton;
	testtime:ton;
	i:UDINT;
	qos:QoS:=2;
	sub1:MQTTSubscribe;
	sub2:MQTTSubscribe;
	sub3:MQTTSubscribe;
	con: BOOL;
	TestLongSubscribe: BOOL;

	//Testtopic:SD_MQTT.TestcaseCheckTopivValid;
	//TestSubscribe:SD_MQTT.TestSubscribe;
	received1: BOOL;
	received2: BOOL;
	received3: BOOL;
	longReceived: BOOL;
	CountSucsess:ARRAY[0..100] OF  ULINT;
	MQTTretain:BOOL:=TRUE;
	enable: BOOL;
	ReceiveData:ARRAY[0..100] OF RECEIVE_PAKET;
	receiveIndex:INT;
	TestLen:UINT;
	SubscribeForBigPaket: BOOL;

		t1:HandleSplitTopic;
	s100:STRING[101]:='1111111111111111111111111111111111111111111111111111111111111111111111111111111111111111111111111111';
	sa:STRING:='abcdefghijklmnopqrstuvwxyz';
	sb:STRING:='ABCDEFGHIJKLMNOPQRSTUVWXYZ';
	sc:STRING:='0123456789';
	sd:STRING:='9876543210';
	splus:STRING:='+';
	ssharp:STRING:='#';
	stest:STRING:='test';
	s1:STRING(64000);
	s2:STRING(64000);
	b1:ARRAY[0..bSize+2]OF BYTE;
	
END_VAR
VAR CONSTANT
	bSize:UDINT := 1024*1024*30;
END_VAR

MQTT_IN_OUT.ClientID :=clientID;
MQTT_IN_OUT.COM_CONFIG.MaxPayloadSize :=50000;
MQTT_IN_OUT.COM_CONFIG.MaxTopicLevels := 200;
//MQTT_IN_OUT.PORT := 1883;
//MQTT_IN_OUT.URL := 'test.mosquitto.org';


{info 'TODO make some nice test cases'}




//testtime(IN:= , PT:= );
testtime(IN:= NOT testtime.Q AND sendTest, PT:= T#50MS);
testTimeBigPublish(IN:= NOT testTimeBigPublish.Q AND testBigPublish, PT:= T#100MS);
testTimeBigPayload(IN:= NOT testTimeBigPayload.Q AND testBigPayload, PT:= T#100MS);
//testtime(IN:= NOT testtime.Q AND sendTest, PT:= T#10S);
IF NOT init THEN
	init := TRUE;
	//Testtopic();
	FOR i := 0 TO 100 DO
		testPublish[i].SetMqttInOut(MQTT_IN_OUT := ADR(MQTT_IN_OUT));
	END_FOR
	FOR i := 0 TO 90 DO
		CommonTypesAndFunctions.concat(s1:= ADR(s1), s2:= ADR(sa));
		CommonTypesAndFunctions.concat(s1:= ADR(s1), s2:= ADR('/'));
		CommonTypesAndFunctions.concat(s1:= ADR(s1), s2:= ADR(sb));
		CommonTypesAndFunctions.concat(s1:= ADR(s1), s2:= ADR('/'));
	END_FOR
	FOR i := 0 TO 10 DO
		CommonTypesAndFunctions.concat(s1:= ADR(s2), s2:= ADR(sc));
		CommonTypesAndFunctions.concat(s1:= ADR(s2), s2:= ADR('/'));
		CommonTypesAndFunctions.concat(s1:= ADR(s2), s2:= ADR(sd));
		CommonTypesAndFunctions.concat(s1:= ADR(s2), s2:= ADR('/'));
	END_FOR
	FOR i := 0 TO bSize DO
		b1[i] := UDINT_TO_BYTE(i);
	END_FOR
	sub1.SetMqttInOut(MQTT_IN_OUT:= ADR(MQTT_IN_OUT));
	sub2.SetMqttInOut(MQTT_IN_OUT:= ADR(MQTT_IN_OUT));
	sub3.SetMqttInOut(MQTT_IN_OUT:= ADR(MQTT_IN_OUT));
	
END_IF

FOR i := 0 TO 20 DO
	CountSucsess[i] := testPublish[i].CountSend;
END_FOR

TestLen := CommonTypesAndFunctions.len(str:= ADR(''));
TestLen := CommonTypesAndFunctions.len(str:= ADR('a'));
TestLen := CommonTypesAndFunctions.len(str:= ADR('aa'));

//	TestSubscribe();
(*
sub1(
	Subscribe:= con, 
	Topic:= ADR(s2), 
	QoSSubscribe:= 2,
	Received => longReceived,
	ExpectingString := TRUE
	 );
sub2(
	Subscribe:= TestLongSubscribe, 
	Topic:= ADR(s1), 
	QoSSubscribe:= 2 ,
	Recieved => received1,
	ExpectingString := TRUE
	 );
sub3(
	Subscribe:= SubscribeForBigPaket, 
	Topic:= ADR('#'), 
	QoSSubscribe:= 2 ,
	Received => received2,
	ExpectingString := FALSE
	 );
IF received1 THEN
	i:=i;
	RecieveData[receiveIndex].MqttPayload := sub1.PayloadString^;
	ReceiveData[receiveIndex].MqttTopic := sub1.TopicOut^;
	receiveIndex := receiveIndex + 1;
	IF receiveIndex > 100 THEN
		receiveIndex := 0;
	END_IF
END_IF*)
testPublish[17](
	Topic:= ADR(s1), 
	Payload:= ADR(b1), 
	QoSIn:= qos, 
	MRetain:= MQTTretain, 
	send := testTimeBigPayload.Q,
	PayloadLength :=  3654,
	PublishAsString := FALSE
	);
testPublish[16](
	Topic:= ADR(s1), 
	PayloadString:= ADR(s2), 
	QoSIn:= qos, 
	MRetain:= MQTTretain, 
	send := testTimeBigPublish.Q, 
	PublishAsString := TRUE
	);
testPublish[0](
	Topic:= ADR('test/topic veryyyyyyyyyyyyyyyyyyyyyyyyyyyyyyyyyyyyyyyyyyyyyyyyyyyyyyyyyyyyyyyyyyyyyyyyyyyyyyyyyyyyyyyyyyyyyyyyyyyyyyyyyyyyyyyyyy big topic/1'), 
	PayloadString:= ADR('test pi1'), 
	QoSIn:= qos, 
	MRetain:= MQTTretain, 
	send := testtime.Q,
	PublishAsString := TRUE 
	);
	
testPublish[1](
	Topic:= ADR('test/topic veryyyyyyyyyyyyyyyyyyyyyyyyyyyyyyyyyyyyyyyyyyyyyyyyyyyyyyyyyyyyyyyyyyyyyyyyyyyyyyyyyyyyyyyyyyyyyyyyyyyyyyyyyyyyyyyyyy big topic/2'), 
	PayloadString:= ADR('test pi2'), 
	QoSIn:= qos, 
	MRetain:= MQTTretain, 
	send := testtime.Q,
	PublishAsString := TRUE 
	);
testPublish[2](
	Topic:= ADR('test/topic veryyyyyyyyyyyyyyyyyyyyyyyyyyyyyyyyyyyyyyyyyyyyyyyyyyyyyyyyyyyyyyyyyyyyyyyyyyyyyyyyyyyyyyyyyyyyyyyyyyyyyyyyyyyyyyyyyy big topic/3'), 
	PayloadString:= ADR('test pi3'), 
	QoSIn:= qos, 
	MRetain:= MQTTretain, 
	send := testtime.Q,
	PublishAsString := TRUE 
	);
testPublish[3](
	Topic:= ADR('test/topic veryyyyyyyyyyyyyyyyyyyyyyyyyyyyyyyyyyyyyyyyyyyyyyyyyyyyyyyyyyyyyyyyyyyyyyyyyyyyyyyyyyyyyyyyyyyyyyyyyyyyyyyyyyyyyyyyyy big topic/4'), 
	PayloadString:= ADR('test pi4'), 
	QoSIn:= qos, 
	MRetain:= MQTTretain, 
	send := testtime.Q, 
	PublishAsString := TRUE
	);
testPublish[4](
	Topic:= ADR('test/topic veryyyyyyyyyyyyyyyyyyyyyyyyyyyyyyyyyyyyyyyyyyyyyyyyyyyyyyyyyyyyyyyyyyyyyyyyyyyyyyyyyyyyyyyyyyyyyyyyyyyyyyyyyyyyyyyyyy big topic/5'), 
	PayloadString:= ADR('test pi5'), 
	QoSIn:= qos, 
	MRetain:= MQTTretain, 
	send := testtime.Q, 
	PublishAsString := TRUE
	);
testPublish[5](
	Topic:= ADR('test/topic veryyyyyyyyyyyyyyyyyyyyyyyyyyyyyyyyyyyyyyyyyyyyyyyyyyyyyyyyyyyyyyyyyyyyyyyyyyyyyyyyyyyyyyyyyyyyyyyyyyyyyyyyyyyyyyyyyy big topic/6'), 
	PayloadString:= ADR('test pi6'), 
	QoSIn:= qos, 
	MRetain:= MQTTretain, 
	send := testtime.Q, 
	PublishAsString := TRUE
	);
testPublish[6](
	Topic:= ADR('test/topic veryyyyyyyyyyyyyyyyyyyyyyyyyyyyyyyyyyyyyyyyyyyyyyyyyyyyyyyyyyyyyyyyyyyyyyyyyyyyyyyyyyyyyyyyyyyyyyyyyyyyyyyyyyyyyyyyyy big topic/7'), 
	PayloadString:= ADR('test pi7'), 
	QoSIn:= qos, 
	MRetain:= MQTTretain, 
	send := testtime.Q, 
	PublishAsString := TRUE
	);
testPublish[7](
	Topic:= ADR('test/topic veryyyyyyyyyyyyyyyyyyyyyyyyyyyyyyyyyyyyyyyyyyyyyyyyyyyyyyyyyyyyyyyyyyyyyyyyyyyyyyyyyyyyyyyyyyyyyyyyyyyyyyyyyyyyyyyyyy big topic/8'), 
	PayloadString:= ADR('test pi8'), 
	QoSIn:= qos, 
	MRetain:= MQTTretain, 
	send := testtime.Q, 
	PublishAsString := TRUE
	);
testPublish[8](
	Topic:= ADR('test/topic veryyyyyyyyyyyyyyyyyyyyyyyyyyyyyyyyyyyyyyyyyyyyyyyyyyyyyyyyyyyyyyyyyyyyyyyyyyyyyyyyyyyyyyyyyyyyyyyyyyyyyyyyyyyyyyyyyy big topic/9'), 
	PayloadString:= ADR('test pi9'), 
	QoSIn:= qos, 
	MRetain:= MQTTretain, 
	send := testtime.Q, 
	PublishAsString := TRUE
	);
testPublish[9](
	Topic:= ADR('test/topic veryyyyyyyyyyyyyyyyyyyyyyyyyyyyyyyyyyyyyyyyyyyyyyyyyyyyyyyyyyyyyyyyyyyyyyyyyyyyyyyyyyyyyyyyyyyyyyyyyyyyyyyyyyyyyyyyyy big topic/10'), 
	PayloadString:= ADR('test pi10'), 
	QoSIn:= qos, 
	MRetain:= MQTTretain, 
	send := testtime.Q, 
	PublishAsString := TRUE
	);
testPublish[10](
	Topic:= ADR('test/topic veryyyyyyyyyyyyyyyyyyyyyyyyyyyyyyyyyyyyyyyyyyyyyyyyyyyyyyyyyyyyyyyyyyyyyyyyyyyyyyyyyyyyyyyyyyyyyyyyyyyyyyyyyyyyyyyyyy big topic/11'), 
	PayloadString:= ADR('test pi11'), 
	QoSIn:= qos, 
	MRetain:= MQTTretain, 
	send := testtime.Q, 
	PublishAsString := TRUE
	);
testPublish[11](
	Topic:= ADR('test/topic veryyyyyyyyyyyyyyyyyyyyyyyyyyyyyyyyyyyyyyyyyyyyyyyyyyyyyyyyyyyyyyyyyyyyyyyyyyyyyyyyyyyyyyyyyyyyyyyyyyyyyyyyyyyyyyyyyy big topic/12'), 
	PayloadString:= ADR('test pi12'), 
	QoSIn:= qos, 
	MRetain:= MQTTretain, 
	send := testtime.Q, 
	PublishAsString := TRUE
	);
testPublish[12](
	Topic:= ADR('test/topic veryyyyyyyyyyyyyyyyyyyyyyyyyyyyyyyyyyyyyyyyyyyyyyyyyyyyyyyyyyyyyyyyyyyyyyyyyyyyyyyyyyyyyyyyyyyyyyyyyyyyyyyyyyyyyyyyyy big topic/13'), 
	PayloadString:= ADR('test pi13'), 
	QoSIn:= qos, 
	MRetain:= MQTTretain, 
	send := testtime.Q, 
	PublishAsString := TRUE
	);
testPublish[13](
	Topic:= ADR('test/topic veryyyyyyyyyyyyyyyyyyyyyyyyyyyyyyyyyyyyyyyyyyyyyyyyyyyyyyyyyyyyyyyyyyyyyyyyyyyyyyyyyyyyyyyyyyyyyyyyyyyyyyyyyyyyyyyyyy big topic/14'), 
	PayloadString:= ADR('test pi14'), 
	QoSIn:= qos, 
	MRetain:= MQTTretain, 
	send := testtime.Q, 
	PublishAsString := TRUE
	);
testPublish[14](
	Topic:= ADR('test/topic veryyyyyyyyyyyyyyyyyyyyyyyyyyyyyyyyyyyyyyyyyyyyyyyyyyyyyyyyyyyyyyyyyyyyyyyyyyyyyyyyyyyyyyyyyyyyyyyyyyyyyyyyyyyyyyyyyy big topic/15'), 
	PayloadString:= ADR('test pi15'), 
	QoSIn:= qos, 
	MRetain:= MQTTretain, 
	send := testtime.Q, 
	PublishAsString := TRUE
	);
testPublish[15](
	Topic:= ADR('test/topic veryyyyyyyyyyyyyyyyyyyyyyyyyyyyyyyyyyyyyyyyyyyyyyyyyyyyyyyyyyyyyyyyyyyyyyyyyyyyyyyyyyyyyyyyyyyyyyyyyyyyyyyyyyyyyyyyyy big topic/16'), 
	PayloadString:= ADR('test pi16'), 
	QoSIn:= qos, 
	MRetain:= MQTTretain, 
	send := testtime.Q, 
	PublishAsString := TRUE
	);






MQTT(
	MQTT_IN_OUT:= MQTT_IN_OUT, 
	ENABLE:= enable, 
	URL:= 'test.mosquitto.org:1883', 
	TIMEOUT:= T#5S, 
	ERROR_C=> ERROR_C, 
	ERROR_T=> ERROR_T);

END_FUNCTION_BLOCK

// MQTT/TestCases/TestMqttTLS
FUNCTION_BLOCK TestMqttTLS
VAR_INPUT
END_VAR
VAR_OUTPUT
END_VAR
VAR
	MQTT:HANDLE_MQTT;
	
	MQTT_IN_OUT:MQTT_IN_OUT;
	ERROR_C:DWORD;
	ERROR_T:BYTE;
	//testPiublish: SD_MQTT.MQTTPublish;
	testPublish: ARRAY[0..100] OF MQTTPublish;
	init:BOOL := FALSE;
	sendTest: BOOL;
	testtime:ton;
	i:UINT;
	qos:QoS:=2;
	sub1:MQTTSubscribe;
	sub2:MQTTSubscribe;
	con: BOOL;
	received: BOOL;
	CountSucsess:ARRAY[0..100] OF  ULINT;
	MQTTretain:BOOL:=TRUE;
	enable: BOOL;
	ReceiveData:ARRAY[0..100] OF RECEIVE_PAKET;
	receiveIndex:INT;
	testTls: BOOL := TRUE;
	
	TLS_CONFIG:CommonTypesAndFunctions.TLS_CONFIG;

END_VAR

MQTT_IN_OUT.ClientID :='testCodesys';
//MQTT_IN_OUT.PORT := 1883;
//MQTT_IN_OUT.URL := 'test.mosquitto.org';

testtime(IN:= NOT testtime.Q AND sendTest, PT:= T#100MS);
//testtime(IN:= NOT testtime.Q AND sendTest, PT:= T#10S);
IF NOT init THEN
	init := TRUE;
	sub1.SetMqttInOut(MQTT_IN_OUT:= ADR(MQTT_IN_OUT));
	sub2.SetMqttInOut(MQTT_IN_OUT:= ADR(MQTT_IN_OUT));
	//Testtopic();
	FOR i := 0 TO 100 DO
		testPublish[i].SetMqttInOut(MQTT_IN_OUT := ADR(MQTT_IN_OUT));
	END_FOR
	
	
	MQTT_IN_OUT.TLS_CONFIG := ADR(TLS_CONFIG);

END_IF

FOR i := 0 TO 20 DO
	CountSucsess[i] := testPublish[i].CountSend;
END_FOR

//	TestSubscribe();
(*
sub1(
	Subscribe:= con, 
	Topic:= ADR('test/#'), 
	QoSSubscribe:= 2 ,
	Received => received,
	ExpectingString := TRUE
	 );
	 
sub2(
	Subscribe:= con, 
	Topic:= ADR('#'), 
	QoSSubscribe:= 2 ,
	Received => received,
	ExpectingString := TRUE
	 );
IF received THEN
	i:=i;
	ReceiveData[receiveIndex].MqttPayload := sub1.PayloadString^;
	ReceiveData[receiveIndex].MqttTopic := sub1.TopicOut^;
	receiveIndex := receiveIndex + 1;
	IF receiveIndex > 100 THEN
		receiveIndex := 0;
	END_IF
END_IF*)
testPublish[0](
	Topic:= ADR('test/topic veryyyyyyyyyyyyyyyyyyyyyyyyyyyyyyyyyyyyyyyyyyyyyyyyyyyyyyyyyyyyyyyyyyyyyyyyyyyyyyyyyyyyyyyyyyyyyyyyyyyyyyyyyyyyyyyyyy big topic/1'), 
	PayloadString:= ADR('test pi1'), 
	QoSIn:= qos, 
	MRetain:= MQTTretain, 
	send := testtime.Q,
	PublishAsString := TRUE 
	);
	
testPublish[1](
	Topic:= ADR('test/topic veryyyyyyyyyyyyyyyyyyyyyyyyyyyyyyyyyyyyyyyyyyyyyyyyyyyyyyyyyyyyyyyyyyyyyyyyyyyyyyyyyyyyyyyyyyyyyyyyyyyyyyyyyyyyyyyyyy big topic/2'), 
	PayloadString:= ADR('test pi2'), 
	QoSIn:= qos, 
	MRetain:= MQTTretain, 
	send := testtime.Q,
	PublishAsString := TRUE 
	);
testPublish[2](
	Topic:= ADR('test/topic veryyyyyyyyyyyyyyyyyyyyyyyyyyyyyyyyyyyyyyyyyyyyyyyyyyyyyyyyyyyyyyyyyyyyyyyyyyyyyyyyyyyyyyyyyyyyyyyyyyyyyyyyyyyyyyyyyy big topic/3'), 
	PayloadString:= ADR('test pi3'), 
	QoSIn:= qos, 
	MRetain:= MQTTretain, 
	send := testtime.Q,
	PublishAsString := TRUE 
	);
testPublish[3](
	Topic:= ADR('test/topic veryyyyyyyyyyyyyyyyyyyyyyyyyyyyyyyyyyyyyyyyyyyyyyyyyyyyyyyyyyyyyyyyyyyyyyyyyyyyyyyyyyyyyyyyyyyyyyyyyyyyyyyyyyyyyyyyyy big topic/4'), 
	PayloadString:= ADR('test pi4'), 
	QoSIn:= qos, 
	MRetain:= MQTTretain, 
	send := testtime.Q, 
	PublishAsString := TRUE
	);
testPublish[4](
	Topic:= ADR('test/topic veryyyyyyyyyyyyyyyyyyyyyyyyyyyyyyyyyyyyyyyyyyyyyyyyyyyyyyyyyyyyyyyyyyyyyyyyyyyyyyyyyyyyyyyyyyyyyyyyyyyyyyyyyyyyyyyyyy big topic/5'), 
	PayloadString:= ADR('test pi5'), 
	QoSIn:= qos, 
	MRetain:= MQTTretain, 
	send := testtime.Q, 
	PublishAsString := TRUE
	);
testPublish[5](
	Topic:= ADR('test/topic veryyyyyyyyyyyyyyyyyyyyyyyyyyyyyyyyyyyyyyyyyyyyyyyyyyyyyyyyyyyyyyyyyyyyyyyyyyyyyyyyyyyyyyyyyyyyyyyyyyyyyyyyyyyyyyyyyy big topic/6'), 
	PayloadString:= ADR('test pi6'), 
	QoSIn:= qos, 
	MRetain:= MQTTretain, 
	send := testtime.Q, 
	PublishAsString := TRUE
	);
testPublish[6](
	Topic:= ADR('test/topic veryyyyyyyyyyyyyyyyyyyyyyyyyyyyyyyyyyyyyyyyyyyyyyyyyyyyyyyyyyyyyyyyyyyyyyyyyyyyyyyyyyyyyyyyyyyyyyyyyyyyyyyyyyyyyyyyyy big topic/7'), 
	PayloadString:= ADR('test pi7'), 
	QoSIn:= qos, 
	MRetain:= MQTTretain, 
	send := testtime.Q, 
	PublishAsString := TRUE
	);
testPublish[7](
	Topic:= ADR('test/topic veryyyyyyyyyyyyyyyyyyyyyyyyyyyyyyyyyyyyyyyyyyyyyyyyyyyyyyyyyyyyyyyyyyyyyyyyyyyyyyyyyyyyyyyyyyyyyyyyyyyyyyyyyyyyyyyyyy big topic/8'), 
	PayloadString:= ADR('test pi8'), 
	QoSIn:= qos, 
	MRetain:= MQTTretain, 
	send := testtime.Q, 
	PublishAsString := TRUE
	);
testPublish[8](
	Topic:= ADR('test/topic veryyyyyyyyyyyyyyyyyyyyyyyyyyyyyyyyyyyyyyyyyyyyyyyyyyyyyyyyyyyyyyyyyyyyyyyyyyyyyyyyyyyyyyyyyyyyyyyyyyyyyyyyyyyyyyyyyy big topic/9'), 
	PayloadString:= ADR('test pi9'), 
	QoSIn:= qos, 
	MRetain:= MQTTretain, 
	send := testtime.Q, 
	PublishAsString := TRUE
	);
testPublish[9](
	Topic:= ADR('test/topic veryyyyyyyyyyyyyyyyyyyyyyyyyyyyyyyyyyyyyyyyyyyyyyyyyyyyyyyyyyyyyyyyyyyyyyyyyyyyyyyyyyyyyyyyyyyyyyyyyyyyyyyyyyyyyyyyyy big topic/10'), 
	PayloadString:= ADR('test pi10'), 
	QoSIn:= qos, 
	MRetain:= MQTTretain, 
	send := testtime.Q, 
	PublishAsString := TRUE
	);
testPublish[10](
	Topic:= ADR('test/topic veryyyyyyyyyyyyyyyyyyyyyyyyyyyyyyyyyyyyyyyyyyyyyyyyyyyyyyyyyyyyyyyyyyyyyyyyyyyyyyyyyyyyyyyyyyyyyyyyyyyyyyyyyyyyyyyyyy big topic/11'), 
	PayloadString:= ADR('test pi11'), 
	QoSIn:= qos, 
	MRetain:= MQTTretain, 
	send := testtime.Q, 
	PublishAsString := TRUE
	);
testPublish[11](
	Topic:= ADR('test/topic veryyyyyyyyyyyyyyyyyyyyyyyyyyyyyyyyyyyyyyyyyyyyyyyyyyyyyyyyyyyyyyyyyyyyyyyyyyyyyyyyyyyyyyyyyyyyyyyyyyyyyyyyyyyyyyyyyy big topic/12'), 
	PayloadString:= ADR('test pi12'), 
	QoSIn:= qos, 
	MRetain:= MQTTretain, 
	send := testtime.Q, 
	PublishAsString := TRUE
	);
testPublish[12](
	Topic:= ADR('test/topic veryyyyyyyyyyyyyyyyyyyyyyyyyyyyyyyyyyyyyyyyyyyyyyyyyyyyyyyyyyyyyyyyyyyyyyyyyyyyyyyyyyyyyyyyyyyyyyyyyyyyyyyyyyyyyyyyyy big topic/13'), 
	PayloadString:= ADR('test pi13'), 
	QoSIn:= qos, 
	MRetain:= MQTTretain, 
	send := testtime.Q, 
	PublishAsString := TRUE
	);
testPublish[13](
	Topic:= ADR('test/topic veryyyyyyyyyyyyyyyyyyyyyyyyyyyyyyyyyyyyyyyyyyyyyyyyyyyyyyyyyyyyyyyyyyyyyyyyyyyyyyyyyyyyyyyyyyyyyyyyyyyyyyyyyyyyyyyyyy big topic/14'), 
	PayloadString:= ADR('test pi14'), 
	QoSIn:= qos, 
	MRetain:= MQTTretain, 
	send := testtime.Q, 
	PublishAsString := TRUE
	);
testPublish[14](
	Topic:= ADR('test/topic veryyyyyyyyyyyyyyyyyyyyyyyyyyyyyyyyyyyyyyyyyyyyyyyyyyyyyyyyyyyyyyyyyyyyyyyyyyyyyyyyyyyyyyyyyyyyyyyyyyyyyyyyyyyyyyyyyy big topic/15'), 
	PayloadString:= ADR('test pi15'), 
	QoSIn:= qos, 
	MRetain:= MQTTretain, 
	send := testtime.Q, 
	PublishAsString := TRUE
	);
testPublish[15](
	Topic:= ADR('test/topic veryyyyyyyyyyyyyyyyyyyyyyyyyyyyyyyyyyyyyyyyyyyyyyyyyyyyyyyyyyyyyyyyyyyyyyyyyyyyyyyyyyyyyyyyyyyyyyyyyyyyyyyyyyyyyyyyyy big topic/16'), 
	PayloadString:= ADR('test pi16'), 
	QoSIn:= qos, 
	MRetain:= MQTTretain, 
	send := testtime.Q, 
	PublishAsString := TRUE
	);




(*
MQTT(
	MQTT_INFO:= MQTT_INFO, 
	MQTT_IN_OUT:= MQTT_IN_OUT, 
	ENABLE:= TRUE, 
	URL:= 'test.mosquitto.org:1883', 
	TIMEOUT:= T#5S, 
	ERROR_C=> ERROR_C, 
	ERROR_T=> ERROR_T);
	*)
	(*
	MQTT(
	MQTT_INFO:= MQTT_INFO, 
	MQTT_IN_OUT:= MQTT_IN_OUT, 
	ENABLE:= enable, 
	URL:= 'localhost:1883', 
	TIMEOUT:= T#5S, 
	ERROR_C=> ERROR_C, 
	ERROR_T=> ERROR_T);
	*)


IF testtls THEN
	
(*
MQTT(
	MQTT_INFO:= MQTT_INFO, 
	MQTT_IN_OUT:= MQTT_IN_OUT, 
	ENABLE:= enable, 
	URL:= 'windows-10-pro:8883', //8883 encryptet, 1883 unencryptet
	TIMEOUT:= T#5S, 
	TLS := TRUE,
	ERROR_C=> ERROR_C, 
	ERROR_T=> ERROR_T);
	*)
	MQTT(
	MQTT_IN_OUT:= MQTT_IN_OUT, 
	ENABLE:= enable, 
	URL:= 'test.mosquitto.org:8883', //8883 encryptet, 1883 unencryptet
	TIMEOUT:= T#5S, 
	TLS := TRUE,
	ERROR_C=> ERROR_C, 
	ERROR_T=> ERROR_T);
	
	

ELSE
MQTT(
	MQTT_IN_OUT:= MQTT_IN_OUT, 
	ENABLE:= enable, 
	URL:= 'test.mosquitto.org:1883', //8883 encryptet, 1883 unencryptet
	TIMEOUT:= T#5S, 
	TLS := FALSE,
	ERROR_C=> ERROR_C, 
	ERROR_T=> ERROR_T);
END_IF

END_FUNCTION_BLOCK

// MQTT/TestCases/TestTopicMatch
FUNCTION_BLOCK TestTopicMatch
VAR_INPUT
END_VAR
VAR_OUTPUT
END_VAR
VAR
	t1:HandleSplitTopic;
	t2:HandleSplitTopic;
	match:TOPIC_MATCH;
	pts:ARRAY[0..20] OF POINTER TO STRING; 
	sp: POINTER TO SPLIT_TOPIC;
	COM_CONFIG: COM_CONFIG;
	dynMemUsage:UDINT;
END_VAR

t1.FullInit(TopicsLevelInit:= 40, SplitElementSizeInit:= 5000, dynMemUsageInit:= ADR(dynMemUsage));
t2.FullInit(TopicsLevelInit:= 40, SplitElementSizeInit:= 5000, dynMemUsageInit:= ADR(dynMemUsage));


t1.NewTopic(in:=ADR('/+/test/#'),test:= TRUE, SizeOfString:= 0);
	sp := t1.GetSplitTopic();
	pts[0] := sp^.Topics[0];
	pts[1] := sp^.Topics[1];
	pts[2] := sp^.Topics[2];
	pts[3] := sp^.Topics[3];
	pts[4] := sp^.Topics[4];
	pts[5] := sp^.Topics[5];
	pts[6] := sp^.Topics[6];
	pts[7] := sp^.Topics[7];
	pts[8] := sp^.Topics[8];
t2.NewTopic(in:=ADR('/rtt/test/tr'),test:= FALSE, SizeOfString:= 0);
	sp := t2.GetSplitTopic();
	pts[10] := sp^.Topics[0];
	pts[11] := sp^.Topics[1];
	pts[12] := sp^.Topics[2];
	pts[13] := sp^.Topics[3];
	pts[14] := sp^.Topics[4];
	pts[15] := sp^.Topics[5];
	pts[16] := sp^.Topics[6];
	pts[17] := sp^.Topics[7];
	pts[18] := sp^.Topics[8];
match := t1.CheckTopicMatchToMe(with:= t2.GetSplitTopic());


//test from MQTT doku
t1.NewTopic(in:=ADR('sport/tennis/+'),test:= TRUE, SizeOfString:= 0);
t2.NewTopic(in:=ADR('sport/tennis/player1'),test:= FALSE, SizeOfString:= 0);
match := t1.CheckTopicMatchToMe(with:= t2.GetSplitTopic()); //match
t2.NewTopic(in:=ADR('sport/tennis/player2'),test:= FALSE, SizeOfString:= 0);
match := t1.CheckTopicMatchToMe(with:= t2.GetSplitTopic());//match
t2.NewTopic(in:=ADR('sport/tennis/player1/ranking'),test:= FALSE, SizeOfString:= 0);
match := t1.CheckTopicMatchToMe(with:= t2.GetSplitTopic());//no match


t1.NewTopic(in:=ADR('sport/+'),test:= TRUE, SizeOfString:= 0);
t2.NewTopic(in:=ADR('sport'),test:= FALSE, SizeOfString:= 0);
match := t1.CheckTopicMatchToMe(with:= t2.GetSplitTopic()); //no match

t2.NewTopic(in:=ADR('sport/'),test:= FALSE, SizeOfString:= 0);
match := t1.CheckTopicMatchToMe(with:= t2.GetSplitTopic()); //match

t1.NewTopic(in:=ADR('+/+'),test:= TRUE, SizeOfString:= 0);
t2.NewTopic(in:=ADR('/finance'),test:= FALSE, SizeOfString:= 0);
match := t1.CheckTopicMatchToMe(with:= t2.GetSplitTopic()); //match

t1.NewTopic(in:=ADR('/+'),test:= TRUE, SizeOfString:= 0);
match := t1.CheckTopicMatchToMe(with:= t2.GetSplitTopic()); //match

t1.NewTopic(in:=ADR('+'),test:= TRUE, SizeOfString:= 0);
match := t1.CheckTopicMatchToMe(with:= t2.GetSplitTopic()); //no match
//just for breakpoint
t1.NewTopic(in:=ADR('+/+'),test:= TRUE, SizeOfString:= 0);

END_FUNCTION_BLOCK

// MQTT/Function Blocks/MQTTValue
FUNCTION_BLOCK MQTTValue
VAR_INPUT
	
	
END_VAR
VAR_OUTPUT
END_VAR
VAR
	Topic:POINTER TO STRING(255);
	ValueName:POINTER TO STRING(255);
	ValuePointer:CommonTypesAndFunctions.ALL_TYPES_UNION_POINTER;
	ValueType : CommonTypesAndFunctions.VAR_TYPES;
	ValueDiff : UINT;
	Value:CommonTypesAndFunctions.ALL_TYPES_UNION;
	InitDone: BOOL;
	Send: BOOL;
	SendDone: BOOL;
	OldValue:CommonTypesAndFunctions.ALL_TYPES_UNION;
	RequestToSend: BOOL;
	 
	Publish:MQTTPublish;
	PayloadTemplate:STRING(255);
	Payload:STRING(255);
	DecimalPlace:INT;
	ValueString:STRING;
	QoS:QoS;
	RetainMqtt: BOOL;
	PowerForReal:UINT;
	MinTime:TIME;
	MinTimeTimer:ton;
	//Start block time of sending
	SendBlock: BOOL;
	PayloadBuild: BOOL;

END_VAR

IF NOT InitDone THEN RETURN; END_IF

publish(
	Topic:= Topic, 
	PayloadString:= ADR(Payload), 
	PublishAsString:= TRUE, 
	QoSIn:= QoS, 
	MRetain:= RetainMqtt, 
	send:= Send, 
	done=> SendDone);


MinTimeTimer(IN:= SendBlock, PT:= MinTime);
IF MinTimeTimer.Q THEN
	SendBlock := FALSE;
END_IF

Value := CommonTypesAndFunctions.GetValueFromPointer(PointerToValue:= ValuePointer, TypeOfValue:= ValueType);
IF NOT SendBlock THEN
	IF CommonTypesAndFunctions.CheckDeltaValue(Value:= Value,
			 TypeOfValue:= ValueType, DeltaVar:= ValueDiff, LastValue:= OldValue,Faktor:= PowerForReal)THEN
		RequestToSend := TRUE;
	END_IF
END_IF
		 
IF RequestToSend AND NOT Send AND NOT SendBlock THEN
	
	Payload := PayloadTemplate;
	ValueString := CommonTypesAndFunctions.GetValueString(VALUE:= Value, TypeOfValue:= ValueType, DecimalPlace:= DecimalPlace);
	CommonTypesAndFunctions.concat(s1:= ADR(Payload), s2:= ADR(ValueString));
	Send := TRUE;
	RequestToSend := FALSE;
END_IF

IF SendDone THEN
	Send := FALSE;
	SendBlock := TRUE;
END_IF

METHOD Init
VAR_INPUT
	//topic name
	Topic:POINTER TO STRING(255);
	//valuve name, placed with ':' bevor value
	ValueName:POINTER TO STRING;
	//pointer to value, can be every datatype
	ValuePointer:CommonTypesAndFunctions.ALL_TYPES_UNION_POINTER;
	//type of the var pointet by ValuePointer
	ValueType : CommonTypesAndFunctions.VAR_TYPES;
	//differenz wich the value have to change bovor it is beeing send. if floting point values it depends on decimals(differen :=1, decimal := 1 --> 0.1 differenz )
	ValueDiff : UINT;
	//decimal places behind comma on floting point values
	DecimalPlace:INT;
	//QoS level of publish
	QoS:QoS;
	//message should be ratained?
	RetainMqtt:BOOL;
	//min Time between publish
	MinTime:TIME;
	//MQTT_IN_OUT
	MQTT_IN_OUT:POINTER TO MQTT_IN_OUT;
END_VAR

VAR

END_VAR
THIS^.Publish.SetMqttInOut(MQTT_IN_OUT:= MQTT_IN_OUT);
THIS^.ValuePointer := ValuePointer;
IF ValueDiff = 0 THEN
	THIS^.ValueDiff := 1;
ELSE
	THIS^.ValueDiff := ValueDiff;	
END_IF

THIS^.Topic := Topic;
THIS^.ValueName := ValueName;
THIS^.ValueType := ValueType;
THIS^.PayloadTemplate := ValueName^;
//don't ad ':' if no name is given
IF NOT THIS^.PayloadTemplate[0] = 0 THEN
	CommonTypesAndFunctions.concat(s1:= ADR(THIS^.PayloadTemplate), s2:= ADR(':'));
END_IF
THIS^.DecimalPlace := DecimalPlace;
InitDone := TRUE;
THIS^.RetainMqtt := RetainMqtt;
THIS^.QoS := QoS;
IF THIS^.ValueType = CommonTypesAndFunctions.VAR_TYPES.LREAL_T OR 
	THIS^.ValueType = CommonTypesAndFunctions.VAR_TYPES.REAL_T THEN
	PowerForReal := TO_UINT(EXPT(10,DecimalPlace));
END_IF
THIS^.MinTime := MinTime;
END_METHOD

END_FUNCTION_BLOCK

// MQTT/TestCases/TestPublishValue
FUNCTION_BLOCK TestPublishValue
VAR_INPUT
END_VAR
VAR_OUTPUT
END_VAR
VAR
	
	MQTT:HANDLE_MQTT;
	
	MQTT_IN_OUT:MQTT_IN_OUT;
	init:BOOL := FALSE;
	sendTest: BOOL;
	TestValue:ARRAY[0..99]OF MQTTValue;
	testtime:ton;
	i:UDINT;
	qos:QoS:=2;
	sub1:MQTTSubscribe;
	Values:ARRAY[0..99]OF CommonTypesAndFunctions.ALL_TYPES_UNION;
	temp1:LREAL;
	tmpPointer:CommonTypesAndFunctions.ALL_TYPES_UNION_POINTER;
	MQTTretain:BOOL:=TRUE;
	enable: BOOL;
	ERROR_C:DWORD;
	ERROR_T:BYTE;
	ValueTime:TIME:=T#5S;
END_VAR

MQTT_IN_OUT.ClientID :='testCodesys';
MQTT_IN_OUT.COM_CONFIG.MaxPayloadSize :=50000;
MQTT_IN_OUT.COM_CONFIG.MaxTopicLevels := 200;
//testtime(IN:= , PT:= );
testtime(IN:= NOT testtime.Q AND sendTest, PT:= T#100MS);

//testtime(IN:= NOT testtime.Q AND sendTest, PT:= T#10S);
IF NOT init THEN
	init := TRUE;
	sub1.SetMqttInOut(MQTT_IN_OUT:= ADR(MQTT_IN_OUT));
	tmpPointer.POINTER_TO_LREAL_T := ADR(temp1);
	TestValue[0].Init(
	Topic:= ADR('Haus/Raum1/Tisch/'), 
	ValueName:= ADR('Temperatur'), 
	ValuePointer:= tmpPointer, 
	ValueType:= CommonTypesAndFunctions.VAR_TYPES.LREAL_T, 
	ValueDiff:= 1, 
	DecimalPlace:= 2, 
	QoS:= qos, 
	RetainMqtt:= MQTTretain,
	MinTime:=ValueTime,
	MQTT_IN_OUT:=ADR(MQTT_IN_OUT));
	
END_IF
TestValue[0]();


MQTT(
	MQTT_IN_OUT:= MQTT_IN_OUT, 
	ENABLE:= enable, 
	URL:= 'test.mosquitto.org:1883', 
	TIMEOUT:= T#5S, 
	ERROR_C=> ERROR_C, 
	ERROR_T=> ERROR_T);

END_FUNCTION_BLOCK

// MQTT/Function Blocks/MQTTState
FUNCTION_BLOCK MQTTState
VAR_INPUT
END_VAR
VAR_OUTPUT
END_VAR
VAR
	State:POINTER TO BOOL;
	Topic:POINTER TO STRING;
	StateName:POINTER TO STRING;
	StateValueOn:POINTER TO STRING;
	StateValueOff:POINTER TO STRING;
	InitDone: BOOL;
	Send: BOOL;
	SendDone: BOOL;
	RequestToSendOn: BOOL;
	RequestToSendOff: BOOL;
	
	Publish:MQTTPublish;
	PayloadTemplate:STRING(255);
	Payload:STRING(255);
	QoS:QoS;
	RetainMqtt: BOOL;
	//SendBlock: BOOL;
	RT:R_TRIG;
	FT:F_TRIG;
END_VAR

{info 'need to check string length!'}
publish(
	Topic:= Topic, 
	PayloadString:= ADR(Payload), 
	PublishAsString:= TRUE, 
	QoSIn:= QoS, 
	MRetain:= RetainMqtt, 
	send:= Send, 
	done=> SendDone);

IF NOT InitDone THEN RETURN; END_IF
RT(CLK:= State^);
FT(CLK:= State^);

IF RT.Q THEN
	RequestToSendOn := TRUE;
END_IF

IF FT.Q THEN
	RequestToSendOff := TRUE;
END_IF

IF RequestToSendOn AND NOT send THEN
	//send on
	send:= TRUE;
	Payload := PayloadTemplate;
	CommonTypesAndFunctions.concat(s1:= ADR(Payload), s2:= StateValueOn);
	RequestToSendOn := FALSE;
END_IF

IF RequestToSendOff AND NOT send THEN
	//send on
	send:= TRUE;
	Payload := PayloadTemplate;
	CommonTypesAndFunctions.concat(s1:= ADR(Payload), s2:= StateValueOff);
	RequestToSendOff := FALSE;
END_IF

IF SendDone THEN
	Send := FALSE;
END_IF

METHOD Init
VAR_INPUT
	//pointer to state
	State:POINTER TO BOOL;
	//topic name
	Topic:POINTER TO STRING;
	//valuve name, placed with ':' bevor value
	StateName:POINTER TO STRING;
	MQTT_IN_OUT:POINTER TO MQTT_IN_OUT; 
	StateValueOn:POINTER TO STRING;
	StateValueOff:POINTER TO STRING;
	//QoS lewvel of publish
	QoS:QoS;
	//message should be ratained?
	RetainMqtt:BOOL;
	
END_VAR

VAR

END_VAR
THIS^.Publish.SetMqttInOut(MQTT_IN_OUT := MQTT_IN_OUT);
THIS^.State := State;
THIS^.Topic := Topic;
THIS^.StateName := StateName;
THIS^.StateValueOff := StateValueOff;
THIS^.StateValueOn := StateValueOn;
THIS^.PayloadTemplate := StateName^;
//don't ad ':' if no name is given
IF NOT THIS^.PayloadTemplate[0] = 0 THEN
	CommonTypesAndFunctions.concat(s1:= ADR(THIS^.PayloadTemplate), s2:= ADR(':'));
ELSE
	PayloadTemplate[0] := 0;
END_IF

InitDone := TRUE;
THIS^.RetainMqtt := RetainMqtt;
THIS^.QoS := QoS;
END_METHOD

END_FUNCTION_BLOCK

// MQTT/Exampels/TestOutOfTheBoxNoTLS
FUNCTION_BLOCK TestOutOfTheBoxNoTLS
VAR_INPUT
	//use this input if you want to test with another broker
	client:STRING:='test.mosquitto.org:1883';//test.mosquitto.org
	
END_VAR
VAR_OUTPUT
END_VAR
VAR
	MQTTClient:HANDLE_MQTT;
	MQTT_IN_OUT:MQTT_IN_OUT;
	publish:MQTTPublish;
	subscribe:MQTTSubscribe;
	ReceiveSubscribeTopic:STRING(255);
	ReceiveSubscribePayloadTick:STRING(255);
	ReceiveSubscribePayloadState:STRING(255);
	State :MQTTState;
	init: BOOL;
	varSend: BOOL;
	timerSend:ton;
	t1:ton;
	t2:ton;
	Payload:STRING;
	//the method PublishReceved() is call when an publsih packet form the broker is received.
	StringCallback:ListStringCallback;
	//the array contains the targets and sub topics for receive
	CallBackTargets:ARRAY[0..1] OF LIST_STRING_CALLBACK_DATA := [(Target:=ADR(ReceiveSubscribePayloadState), SubTopic:= ADR('State')),
																(Target:=ADR(ReceiveSubscribePayloadTick), SubTopic:= ADR('Tick'))];
END_VAR

//here init is done
IF NOT init THEN
	init := TRUE;
	MQTT_IN_OUT.ClientID := CONCAT('CodesysMqtt',TO_STRING(TICKS.GetTick(xDummy:= TRUE)));
	publish.SetMqttInOut(MQTT_IN_OUT:= ADR(MQTT_IN_OUT));
	subscribe.SetMqttInOut(MQTT_IN_OUT:= ADR(MQTT_IN_OUT));
	//init state FB, so you only have to call state();without parameters... 
	State.Init(
	State:= ADR(t1.Q), 
	Topic:= ADR('CODESYS-MQTT-BY-SD/State'), 
	StateName:= ADR(''), 
	StateValueOn:= ADR('On'), 
	StateValueOff:= ADR('Off'), 
	QoS:= QoS.ExactlyOnce, 
	RetainMqtt:= TRUE,
	MQTT_IN_OUT:= ADR(MQTT_IN_OUT));
	StringCallback.InitAsSplitTopic(ListData := ADR(CallBackTargets), LengthOfData:= 2);

END_IF
//timer for repeating packets
timerSend(in := NOT varSend, PT := T#2S);
varSend := timerSend.Q; 
t1(IN:= NOT t2.Q, PT:= T#1S, );
t2(IN:= t1.Q, PT:= T#1S, );
//call of MQTT client
MQTTClient( 
	MQTT_IN_OUT:= MQTT_IN_OUT, 
	ENABLE:= TRUE, 
	URL:= client, 
	TIMEOUT:= T#5S, 
	TLS:= FALSE);
//build payload
IF varSend THEN
	Payload:= TO_STRING(TICKS.GetTick(xDummy:= TRUE));
END_IF
//Publish Payload
publish(
	Topic:= ADR('CODESYS-MQTT-BY-SD/Tick'), 
	PayloadString:= ADR(Payload), 
	PublishAsString:= TRUE, 
	QoSIn:= QoS.ExactlyOnce, 
	MRetain:= TRUE, 
	send:= varSend);
//Subscribe to topic
subscribe(
	Subscribe:= TRUE, 
	Topic:= ADR('CODESYS-MQTT-BY-SD/#'), 
	QoSSubscribe:= QoS.ExactlyOnce, 
	ExpectingString:= TRUE,
	Callback:= StringCallback);


//call of state FB
State();

END_FUNCTION_BLOCK

// MQTT/Exampels/TestOutOfTheBoxTLS
FUNCTION_BLOCK TestOutOfTheBoxTLS
VAR_INPUT
	//use this input if you want to test with another broker
	client:STRING:='test.mosquitto.org:8883';//test.mosquitto.org
	
END_VAR
VAR_OUTPUT
END_VAR
VAR
	MQTTClient:HANDLE_MQTT;
	MQTT_IN_OUT:MQTT_IN_OUT;
	publish:MQTTPublish;
	subscribe:MQTTSubscribe;
	ReceiveSubscribeTopic:STRING(255);
	ReceiveSubscribePayloadTick:STRING(255);
	ReceiveSubscribePayloadState:STRING(255);
	State :MQTTState;
	init: BOOL;
	varSend: BOOL;
	timerSend:ton;
	t1:ton;
	t2:ton;
	Payload:STRING;
	//the method PublishReceved() is call when an publsih packet form the broker is received.
	StringCallback:ListStringCallback;
	//the array contains the targets and sub topics for receive
	CallBackTargets:ARRAY[0..1] OF LIST_STRING_CALLBACK_DATA := [(Target:=ADR(ReceiveSubscribePayloadState), SubTopic:= ADR('State')),
																(Target:=ADR(ReceiveSubscribePayloadTick), SubTopic:= ADR('Tick'))];
	TLS_CONFIG:CommonTypesAndFunctions.TLS_CONFIG;
	
END_VAR

//here init is done
IF NOT init THEN
	init := TRUE;
	MQTT_IN_OUT.ClientID := CONCAT('CodesysMqtt',TO_STRING(TICKS.GetTick(xDummy:= TRUE)));
	publish.SetMqttInOut(MQTT_IN_OUT:= ADR(MQTT_IN_OUT));
	subscribe.SetMqttInOut(MQTT_IN_OUT:= ADR(MQTT_IN_OUT));
	//init state FB, so you only have to call state();without parameters... 
	State.Init(
	State:= ADR(t1.Q), 
	Topic:= ADR('CODESYS-MQTT-BY-SD/State'), 
	StateName:= ADR(''), 
	StateValueOn:= ADR('On'), 
	StateValueOff:= ADR('Off'), 
	QoS:= QoS.ExactlyOnce, 
	RetainMqtt:= TRUE,
	MQTT_IN_OUT:= ADR(MQTT_IN_OUT));
	StringCallback.InitAsSplitTopic(ListData := ADR(CallBackTargets), LengthOfData:= 2);
	MQTT_IN_OUT.TLS_CONFIG := ADR(TLS_CONFIG);
END_IF
//timer for repeating packets
timerSend(in := NOT varSend, PT := T#2S);
varSend := timerSend.Q; 
t1(IN:= NOT t2.Q, PT:= T#1S, );
t2(IN:= t1.Q, PT:= T#1S, );
//call of MQTT client
MQTTClient( 
	MQTT_IN_OUT:= MQTT_IN_OUT, 
	ENABLE:= TRUE, 
	URL:= client, 
	TIMEOUT:= T#5S, 
	TLS:= TRUE);
//build payload
IF varSend THEN
	Payload:= TO_STRING(TICKS.GetTick(xDummy:= TRUE));
END_IF
//Publish Payload
publish(
	Topic:= ADR('CODESYS-MQTT-BY-SD/Tick'), 
	PayloadString:= ADR(Payload), 
	PublishAsString:= TRUE, 
	QoSIn:= QoS.ExactlyOnce, 
	MRetain:= TRUE, 
	send:= varSend);
//Subscribe to topic	
subscribe(
	Subscribe:= TRUE, 
	Topic:= ADR('CODESYS-MQTT-BY-SD/#'), 
	QoSSubscribe:= QoS.ExactlyOnce, 
	ExpectingString:= TRUE,
	Callback:= StringCallback);


//call of state FB
State();

END_FUNCTION_BLOCK

// MQTT/TestCases/testHighReceive
FUNCTION_BLOCK testHighReceive
VAR_INPUT
	topics:UINT:=TEST_TOPICS;
	broker:STRING:='test.mosquitto.org:1883';
	addTopic:STRING(200);
	repeatTime : TIME := T#60S;
END_VAR
VAR_OUTPUT
END_VAR
VAR
	MQTT:HANDLE_MQTT;
	
	send:HighLoadPublish;
	sendWork: BOOL;
	PayloadTarget:POINTER TO POINTER TO STRING;
	subs:MQTTSubscribe;
	MQTT_IN_OUT:MQTT_IN_OUT;
	tNewRun:TON;
	init: BOOL;
	i:UINT;
	testPayload:ARRAY[0..TOPICS_MAX]OF STRING;
	testPayloadPointer:ARRAY[0..TOPICS_MAX]OF POINTER TO STRING;
	emptyString:STRING :='';
	pointerToEmptyString : POINTER TO STRING := ADR(emptyString);
	testTopics:ARRAY[0..TOPICS_MAX]OF STRING(255);
	testTopicsPointer:ARRAY[0..TOPICS_MAX]OF POINTER TO STRING;
	
	compareTopic:ARRAY[0..TOPICS_MAX]OF STRING(255);
	testPayloadReceive:ARRAY[0..TOPICS_MAX]OF STRING;
	PayloadReceiveValue:ARRAY[0..TOPICS_MAX]OF STRING(255);
	SplitChar:STRING:='=';
	tmpString:STRING;
	step:INT;
	topic:STRING(255);
	payload:STRING(255);
	sendPublish: BOOL;
	subscribe: BOOL;
	noData: BOOL;
	nextRun: BOOL;
	ListCallback:ListStringCallback;
	CallbackData:ARRAY[0..TOPICS_MAX] OF LIST_STRING_CALLBACK_DATA;
	PayloadFix: BOOL;

END_VAR
VAR CONSTANT
	TEST_TOPICS:UINT:= 200;
	TOPICS_MAX:UINT:=10000;
END_VAR

IF NOT init THEN
	init := TRUE;
	subs.SetMqttInOut(MQTT_IN_OUT:= ADR(MQTT_IN_OUT)); 
	//Testtopic();
	FOR i := 0 TO topics - 1 DO
		tmpString := UINT_TO_STRING(i);
		testTopics[i] := 'RetainTopicSD/Topic:';
		CommonTypesAndFunctions.concat(s1:= ADR(testTopics[i]), s2:= ADR(addTopic));
		CommonTypesAndFunctions.concat(s1:= ADR(testTopics[i]), s2:= ADR(tmpString));
		testTopicsPointer[i] := ADR(testTopics[i]);
		testPayloadPointer[i] := ADR(testPayload[i]);
		//CommonTypesAndFunctions.concat(s1:= ADR(testTopics[i]), s2:= ADR('/'));
		testPayload[i] := tmpString;
		compareTopic[i] :='Topic:';
		CommonTypesAndFunctions.concat(s1:= ADR(compareTopic[i]), s2:= ADR(addTopic));
		CommonTypesAndFunctions.concat(s1:= ADR(compareTopic[i]), s2:= ADR(tmpString));
		
		//compareTopic[i] := tmpString;
		CallbackData[i].SubTopic := ADR(compareTopic[i]);
		CallbackData[i].Target := ADR(testPayloadReceive[i]);
	END_FOR
	ListCallback.InitAsSplitTopic(ListData:= ADR(CallbackData[0]), LengthOfData:= i);
END_IF
IF topics >= TOPICS_MAX THEN
	topics := TOPICS_MAX;
END_IF

send(
	ClientID:= 'SendHighReceive test', 
	Topic:= ADR(testTopicsPointer), 
	TopicFix:= FALSE, 
	payload:= PayloadTarget, 
	PayloadFix := PayloadFix,
	CountArray:= topics, 
	UsedPublishFbs:= 48, 
	working:= sendWork, 
	broker:= broker, 
	QoS:= QoS.ExactlyOnce, 
	RetainIn:= TRUE);
subs(
	Subscribe:= subscribe, 
	Topic:= ADR('RetainTopicSD/#'), 
	QoSSubscribe:= QoS.ExactlyOnce, 
	ExpectingString:= TRUE,
	Callback := ListCallback);
	

MQTT(
	MQTT_IN_OUT:= MQTT_IN_OUT, 
	ENABLE:= TRUE, 
	URL:= broker, 
	TIMEOUT:= T#5S, 
	TLS:= FALSE);
IF NOT MQTT_IN_OUT.BROKER_CONNECTED THEN
	step := 0;
END_IF
	
CASE step OF
	0: 	step := 1;
		
		FOR i := 0 TO topics - 1 DO
			testPayloadReceive[i] := '';
		END_FOR
	1: IF MQTT_IN_OUT.BROKER_CONNECTED THEN
			step:= 10;
			PayloadTarget := ADR(testPayloadPointer); 
			sendWork := TRUE;
			PayloadFix := FALSE;
		END_IF
	10: //publish all data
		IF send.finished THEN
			sendWork := FALSE;
			step := 30; 
			
		END_IF
	
	30: subscribe := TRUE;
		step := 40;
		
	40: // wait to receive all topics
		noData := FALSE;
		FOR i := 0 TO topics - 1 DO
			IF testPayloadReceive[i] <> testPayload[i] THEN
				noData := TRUE;
			END_IF
		END_FOR
		IF NOT noData THEN
			step := 50; 
		END_IF 
		//unsubscripe
	50: subscribe := FALSE;
		step := 52;
		PayloadTarget := pointerToEmptyString; 
		//cleanup receive buffer
		FOR i := 0 TO topics - 1 DO
			testPayloadReceive[i] :='';
		END_FOR
		sendWork := TRUE;
		PayloadFix := TRUE;
	52: //discharge retain messages from broker
		IF send.finished  THEN
			sendWork := FALSE;
			step := 60;
		END_IF
	
	60:
		IF nextRun OR tNewRun.Q THEN 
			nextRun := FALSE;
			step := 0;
		END_IF
END_CASE

tNewRun(in := step = 60,PT:= repeatTime);

END_FUNCTION_BLOCK

// MQTT/TestCases/HighLoadPublish
FUNCTION_BLOCK HighLoadPublish
VAR_INPUT
	ClientID:STRING(255) := 'TestHighReceive/Topic';
	Topic:POINTER TO POINTER TO STRING;
	TopicFix: BOOL;
	payload:POINTER TO POINTER TO STRING;
	PayloadFix: BOOL;

	CountArray:UINT;
	UsedPublishFbs:UINT;
	//set to high to work, low to stop....
	working: BOOL;
	broker:STRING(255);
	QoS:QoS;
	RetainIn:BOOL;
END_VAR
VAR_OUTPUT
	finished: BOOL;
END_VAR
VAR
	i:UINT;
	Publishs:ARRAY[0..MyConstants.IN_OUT_SLOTS_SIZE] OF MQTTPublish;	
	PublishSendBools:ARRAY[0..MyConstants.IN_OUT_SLOTS_SIZE] OF BOOL;
	PublishSendFree:ARRAY[0..MyConstants.IN_OUT_SLOTS_SIZE] OF BOOL := [MyConstants.IN_OUT_SLOTS_SIZE(TRUE)];
	PublishTopicStore:ARRAY[0..MyConstants.IN_OUT_SLOTS_SIZE] OF POINTER TO STRING;
	PublishPayloadStore:ARRAY[0..MyConstants.IN_OUT_SLOTS_SIZE] OF POINTER TO STRING;
	MQTT:HANDLE_MQTT;
	
	init: BOOL;
	MQTT_IN_OUT:MQTT_IN_OUT;
	LastPublished: UINT;;
	start:R_TRIG;
	
	doPublish: BOOL;

	
END_VAR

IF NOT init THEN
	init := TRUE;
	MQTT_IN_OUT.ClientID := ClientID; 
	FOR i := 0 TO UsedPublishFbs - 1 DO
		
	Publishs[i].SetMqttInOut(MQTT_IN_OUT := ADR(MQTT_IN_OUT));
	END_FOR
END_IF

doPublish := working AND MQTT_IN_OUT.BROKER_CONNECTED;

IF NOT doPublish THEN
	LastPublished := 0;
	FOR i := 0 TO UsedPublishFbs - 1 DO
		PublishSendBools[i] := FALSE;
		Publishs[i](
	send:= PublishSendBools[i]);
	PublishSendFree[i] := TRUE;
	END_FOR
	
END_IF

MQTT(
	MQTT_IN_OUT:= MQTT_IN_OUT, 
	ENABLE:= TRUE, 
	URL:= broker, 
	TIMEOUT:= T#5S, 
	TLS:= FALSE);
start(CLK := working);

IF start.Q THEN
	finished := FALSE;

END_IF
IF doPublish THEN

	FOR i := 0 TO UsedPublishFbs - 1 DO
		
		IF PublishSendFree[i] AND NOT finished THEN
			PublishSendFree[i] := FALSE;
			
			//get next element
			IF LastPublished >= CountArray THEN
				finished := TRUE;
	
			ELSE
				IF TopicFix THEN
					PublishTopicStore[i] := Topic;
				ELSE
					PublishTopicStore[i] := Topic[LastPublished];	
				END_IF
				
				IF PayloadFix THEN
					PublishPayloadStore[i] := Payload;
				ELSE
					PublishPayloadStore[i] := Payload[LastPublished];	
				END_IF
				
				PublishSendBools[i] := TRUE;
			END_IF
			LastPublished := LastPublished + 1;
			
		END_IF	
		
			Publishs[i](
		Topic:=PublishTopicStore[i], 
		PayloadString:= PublishPayloadStore[i], 
		PublishAsString:= TRUE, 
		QoSIn:= QoS, 
		MRetain:= RetainIn, 
		send:= PublishSendBools[i]);
		IF Publishs[i].done THEN 
			PublishSendFree[i] := TRUE;
		END_IF
		IF Publishs[i].sendActive THEN
			PublishSendBools[i] := FALSE;
		END_IF
	END_FOR
	
END_IF

END_FUNCTION_BLOCK

// MQTT/Function/InitMQTTValue
FUNCTION InitMQTTValue : bool
VAR_INPUT
DataArray:POINTER TO CommonTypesAndFunctions.PWConfigs;
CountOfArray:UINT;
ValueToMQTTArray:POINTER TO MQTTValue;
MQTT_IN_OUT: POINTER TO MQTT_IN_OUT;
END_VAR
VAR
	i:UINT;
END_VAR

FOR i := 0 TO CountOfArray - 1 DO
	IF DataArray[i].NeedsMQTT THEN
		ValueToMQTTArray[i].Init(
			Topic:= DataArray[i].MQTTTopic, 
			ValueName:= DataArray[i].MQTTName, 
			ValuePointer:= DataArray[i].PointerTo, 
			ValueType:= DataArray[i].ValueType, 
			ValueDiff:= DataArray[i].MQTTDiff, 
			DecimalPlace:= DataArray[i].MQTTDezimal, 
			QoS:= DataArray[i].MQTTQoS, 
			RetainMqtt:= DataArray[i].MQTTRetain, 
			MinTime:= DataArray[i].MQTTTime,
			MQTT_IN_OUT:= MQTT_IN_OUT);
	END_IF
END_FOR

END_FUNCTION

// MQTT/Function Blocks/MQTTPushover
FUNCTION_BLOCK MQTTPushover
VAR_INPUT
	Data:POINTER TO PUSHOVER_DATA;
	MQTT_IN_OUT:POINTER TO MQTT_IN_OUT;
	CountData:UINT;
	MQTTTopic:POINTER TO STRING;
END_VAR
VAR_OUTPUT
END_VAR
VAR
	i:UINT;
	HaveToPush:BOOL;
	 
	Publish:MQTTPublish;
	init:BOOL;
	PushedElement:UINT;
	SendFree: BOOL;
	// at least one message to push
	hit: BOOL;
	hitIndex:UINT;
	(*build like 'Topic(n(x)):x, Payload(n(x):x, Prio:x, Sound:x'  *)
	SendString:STRING(500);
	tmpString:STRING;
END_VAR

IF NOT init THEN
	
	init := TRUE;
	Publish.SetMqttInOut(MQTT_IN_OUT:= MQTT_IN_OUT);
END_IF
hit := FALSE;
HaveToPush := FALSE;
FOR i := 0 TO CountData - 1 DO
	IF Data[i].IsConfig THEN
		Data[i].R_T(CLK:=Data[i].Trigger^ XOR Data[i].Negate);
		IF Data[i].R_T.Q THEN
			Data[i].NeedToPush := TRUE;
		END_IF
		IF Data[i].NeedToPush THEN
			HaveToPush := TRUE;
		END_IF
		IF HaveToPush and NOT hit THEN
			hit := TRUE;
			hitIndex := i;
		END_IF
	END_IF
END_FOR

IF Publish.done THEN
	SendFree := TRUE;
END_IF


IF HaveToPush AND SendFree THEN
	SendFree := FALSE;
	//now build message
	SendString := 'Topic(';
	//add topic length
	tmpString := TO_STRING(len(Data[hitIndex].Topic^));
 	CommonTypesAndFunctions.concat(s1:= ADR(SendString), S2:=ADR(tmpString));
	//add '):'
	CommonTypesAndFunctions.concat(s1:= ADR(SendString), S2:=ADR('):'));
	//add topic
	CommonTypesAndFunctions.concat(s1:= ADR(SendString), S2:=Data[hitIndex].Topic);
	//add fixtext
	CommonTypesAndFunctions.concat(s1:= ADR(SendString), S2:=ADR(', Payload('));
	//add payload length
	tmpString := TO_STRING(len(Data[hitIndex].Payload^));
 	CommonTypesAndFunctions.concat(s1:= ADR(SendString), S2:=ADR(tmpString));
	//add '):'
	CommonTypesAndFunctions.concat(s1:= ADR(SendString), S2:=ADR('):'));
	//add topic
	CommonTypesAndFunctions.concat(s1:= ADR(SendString), S2:=Data[hitIndex].Payload);
	//add fixtext
	CommonTypesAndFunctions.concat(s1:= ADR(SendString), S2:=ADR(', Prio:'));
	//add prio
	tmpString := TO_STRING(Data[hitIndex].Prio);
 	CommonTypesAndFunctions.concat(s1:= ADR(SendString), S2:=ADR(tmpString));
	//add fixtext
	CommonTypesAndFunctions.concat(s1:= ADR(SendString), S2:=ADR(', Sound:'));
	//add prio
	tmpString := TO_STRING(Data[hitIndex].Sound);
 	CommonTypesAndFunctions.concat(s1:= ADR(SendString), S2:=ADR(tmpString));
	//done
	Data[hitIndex].NeedToPush := FALSE;
	//now send
	
END_IF

Publish(
	Topic:= MQTTTopic, 
	PayloadString:= adr(SendString), 
	PublishAsString:= TRUE, 
	QoSIn:= QoS.ExactlyOnce, 
	MRetain:= true, 
	send:= NOT SendFree);

END_FUNCTION_BLOCK

// MQTT/Function Blocks/CallbackFBs/SingelCallbacks/SingelStringCallback
FUNCTION_BLOCK SingelStringCallback IMPLEMENTS MQTT_SUBSCRIBE_CALLBACK
VAR_INPUT
END_VAR
VAR_OUTPUT
	//data was received, you have to reset this bit after checking!
	received: BOOL;
END_VAR
VAR
	MyPayload : POINTER TO STRING;
	MyTopic : POINTER TO STRING;
END_VAR

METHOD PublishReceived : BOOL
VAR_INPUT
	//Collection of received Data
	Data:CALLBACK_DATA;

END_VAR
MEM.MemMove(pSource:= Data.PayloadString, pDestination:= MyPayload, uiNumberOfBytes:= TO_UINT(data.PayloadSize + 1));
MEM.MemMove(pSource:= Data.TopicOut, pDestination:= MyTopic, uiNumberOfBytes:= CommonTypesAndFunctions.len(Data.TopicOut) + 1);

received := TRUE;
END_METHOD

METHOD Init : BOOL
VAR_INPUT
	payload:POINTER TO STRING;
	topic:POINTER TO STRING;
END_VAR
MyTopic := topic;
MyPayload := payload;
END_METHOD

METHOD ResetReceived : BOOL
VAR_INPUT
END_VAR
received := FALSE;
END_METHOD

END_FUNCTION_BLOCK

// MQTT/Function Blocks/CallbackFBs/SingelCallbacks/AllValuesCallback
(*
this FB expects all values as a string, binary receive is not suported...
Payload content is only value, no description, no special characters...
*)
FUNCTION_BLOCK AllValuesCallback IMPLEMENTS MQTT_SUBSCRIBE_CALLBACK
VAR_INPUT
END_VAR
VAR_OUTPUT
	//data was received, you have to reset this bit after checking!
	received: BOOL;

END_VAR
VAR
	VarType:CommonTypesAndFunctions.VAR_TYPES;
	MyTarget:CommonTypesAndFunctions.ALL_TYPES_UNION_POINTER;
END_VAR

METHOD PublishReceived : BOOL
VAR_INPUT
	//Collection of received Data
	Data:CALLBACK_DATA;

END_VAR
CommonTypesAndFunctions.GetValueFromStringPt(TypeOfValue:= VarType,Target:= MyTarget, str:= DATA.PayloadString);

received := TRUE;
END_METHOD

METHOD Init : BOOL
VAR_INPUT
	SetType:CommonTypesAndFunctions.VAR_TYPES;
	Target:CommonTypesAndFunctions.ALL_TYPES_UNION_POINTER;
END_VAR
VarType := SetType;
MyTarget := Target;
END_METHOD

METHOD ResetReceived : BOOL
VAR_INPUT
END_VAR
received := FALSE;
END_METHOD

END_FUNCTION_BLOCK

// MQTT/Function Blocks/CallbackFBs/ListCallbacks/ListAllValuesCallback
(*
this FB expects all values as a string, binary receive is not suported...
Payload content is only value, no description, no special characters...
*)
FUNCTION_BLOCK ListAllValuesCallback IMPLEMENTS MQTT_SUBSCRIBE_CALLBACK
VAR_INPUT
END_VAR
VAR_OUTPUT
END_VAR
VAR
	MyListData:POINTER TO LIST_ALLVALUES_CALLBACK_DATA;
	MyLengthOfData:ULINT;
	ListSplitTopic:BOOL;
	ListSplitPayload:BOOL;
	SplitCharPayload:BYTE;
END_VAR

METHOD PublishReceived : BOOL
VAR_INPUT
	//Collection of received Data
	Data:CALLBACK_DATA;
END_VAR

VAR
	i:ULINT;
	StrPt:POINTER TO STRING;
END_VAR
IF ListSplitTopic THEN
	//now search the right topic 
	FOR i := 0 TO MyLengthOfData - 1 DO
		IF CommonTypesAndFunctions.StrEquals(str1:= Data.TopicOutSplit^.Topics[Data.TopicOutSplit^.ValidFields - 1], str2:= MyListData[i].SubTopic) THEN
			CommonTypesAndFunctions.GetValueFromStringPt(TypeOfValue:= MyListData[i].VarTYPE ,Target:= MyListData[i].Target, str:= DATA.PayloadString);
		END_IF
	END_FOR
END_IF
IF ListSplitPayload THEN
	FOR i := 0 TO MyLengthOfData - 1 DO
		IF CommonTypesAndFunctions.StrEqualsAtStartWithDelimiter(str1:= MyListData[i].SubTopic, str2:= Data.PayloadString, delimiter:= SplitCharPayload) THEN
			//now search split char
			StrPt := Data.PayloadString;
			StrPt := StrPt + TO_DWORD(CommonTypesAndFunctions.find(str1 := StrPt, str2:= ADR(SplitCharPayload))) + 1;
			
			CommonTypesAndFunctions.GetValueFromStringPt(TypeOfValue:= MyListData[i].VarTYPE ,Target:= MyListData[i].Target, str:= StrPt);
		END_IF
	END_FOR
	
END_IF
END_METHOD

METHOD InitAsSplitTopic : BOOL
VAR_INPUT
	Data:POINTER TO LIST_ALLVALUES_CALLBACK_DATA;
	//Count of List Data
	LengthOfData:ULINT;
END_VAR
MyListData := Data;
MyLengthOfData := LengthOfData;
ListSplitTopic := TRUE;
ListSplitPayload := FALSE;
END_METHOD

(*inits FB, callback methoth then checks if the payload ist the same in the first characters as in the template
make sure to receive a string payload!
*)
METHOD InitAsSplitPayload : BOOL
VAR_INPUT
	Data:POINTER TO LIST_ALLVALUES_CALLBACK_DATA;
	//Count of List Data
	LengthOfData:ULINT;
	//spliting character
	SplitChar:BYTE;
END_VAR
MyListData :=Data;
MyLengthOfData := LengthOfData;
ListSplitTopic := FALSE;
ListSplitPayload := TRUE;
SplitCharPayload := SplitChar;
END_METHOD

END_FUNCTION_BLOCK

// MQTT/TestCases/testHighReceiveSplitPayload
FUNCTION_BLOCK testHighReceiveSplitPayload
VAR_INPUT
	Count:UINT:=TEST_TOPICS;
	broker:STRING:='test.mosquitto.org:1883';
	addTopic:STRING(200);
	repeatTime:TIME:=T#1M;
END_VAR
VAR_OUTPUT
END_VAR
VAR
	MQTT_RECEIVE:HANDLE_MQTT;
	
	
	subs:MQTTSubscribe;
	MQTT_IN_OUT_RECEIVE:MQTT_IN_OUT;
	tNewRun:TON;
	init: BOOL;
	i:UINT;
	//testTopics:ARRAY[0..TOPICS_MAX] OF STRING(255);
	testTopic:STRING:='SD_MQTT/TEST_PAYLOAD/PAYLOAD';
	testPayloadString:ARRAY[0..TOPICS_MAX]OF STRING(255);
	splitChar:STRING := '=';
	PayloadPrefix:STRING := 'Output';
	comparePayload:ARRAY[0..TOPICS_MAX]OF STRING(255);
	
	SendPayloadStorePointerArray:ARRAY[0..TOPICS_MAX] OF POINTER TO STRING;
	ReceivePayloadStore:ARRAY[0..TOPICS_MAX] OF LINT;
	SendPayloadStore:ARRAY[0..TOPICS_MAX] OF LINT;
	
	tmpString:STRING;
	tmpString2:STRING;
	step:UINT;
	subscribe: BOOL;

	HighSendPublish:HighLoadPublish;
	
	runPublishWorker: BOOL;

	
	noData: BOOL;
	nextRun: BOOL;
	ListCallback:ListAllValuesCallback;
	CallbackData:ARRAY[0..TOPICS_MAX] OF LIST_ALLVALUES_CALLBACK_DATA;
END_VAR
VAR CONSTANT
	TEST_TOPICS:UINT:= 200;
	TOPICS_MAX:UINT:=10000;
END_VAR

IF NOT init THEN
	init := TRUE;
	MQTT_IN_OUT_RECEIVE.ClientID := 'Test Client Receive';
	subs.SetMqttInOut(MQTT_IN_OUT:= ADR(MQTT_IN_OUT_RECEIVE)); 
	//Testtopic();
	FOR i := 0 TO Count - 1 DO

		tmpString := PayloadPrefix;
		tmpString2 := UINT_TO_STRING(i);
		CommonTypesAndFunctions.concat(s1:= ADR(tmpString), s2:= ADR(tmpString2));
		//finished building compare payload
		comparePayload[i] := tmpString;
		CommonTypesAndFunctions.concat(s1:= ADR(tmpString), s2:= ADR(splitChar));
		SendPayloadStore[i] := i + 22;
		tmpString2 := TO_STRING(SendPayloadStore[i]);
		CommonTypesAndFunctions.concat(s1:= ADR(tmpString), s2:= ADR(tmpString2));
		//CommonTypesAndFunctions.concat(s1:= ADR(tmpString), s2:= ADR(splitChar));
		
		testPayloadString[i] := tmpString; 
		
		//compareTopic[i] := tmpString;
		CallbackData[i].SubTopic := ADR(comparePayload[i]);
		CallbackData[i].Target.POINTER_TO_LINT_T := ADR(ReceivePayloadStore[i]);
		CallbackData[i].VarTYPE := CommonTypesAndFunctions.VAR_TYPES.LINT_T;
		SendPayloadStorePointerArray[i] := ADR(testPayloadString[i]);
	END_FOR
	ListCallback.InitAsSplitPayload(Data:= ADR(CallbackData[0]), LengthOfData:= i, SplitChar:= CommonTypesAndFunctions.GetChar(splitChar));
END_IF
IF Count >= TOPICS_MAX THEN
	Count := TOPICS_MAX;
END_IF

subs(
	Subscribe:= subscribe, 
	Topic:= ADR(testTopic), 
	QoSSubscribe:= QoS.ExactlyOnce, 
	ExpectingString:= TRUE,
	Callback := ListCallback);
	
MQTT_RECEIVE(
	MQTT_IN_OUT:= MQTT_IN_OUT_RECEIVE, 
	ENABLE:= TRUE, 
	URL:= broker, 
	TIMEOUT:= T#5S, 
	TLS:= FALSE);
IF NOT MQTT_IN_OUT_RECEIVE.BROKER_CONNECTED THEN
	step := 0;
END_IF
	
HighSendPublish(
	ClientID:= 'HighSendClient', 
	Topic:= ADR(testTopic), 
	TopicFix:= TRUE, 
	payload:= ADR(SendPayloadStorePointerArray), 
	CountArray:= Count, 
	UsedPublishFbs:= 49, 
	working:= runPublishWorker, 
	broker:= broker, 
	QoS:= QoS.ExactlyOnce, 
	RetainIn:= FALSE);


CASE step OF
	0: 	step := 1;
		FOR i := 0 TO Count - 1 DO
			ReceivePayloadStore[i] := 0;
		END_FOR
	1: IF MQTT_IN_OUT_RECEIVE.BROKER_CONNECTED THEN
			step:= 5;
			//subscribe
			subscribe := TRUE;
		END_IF
	5: //wait for subscribe
		IF subs.SubscribeDone THEN
			step:= 10;
		END_IF
		 
	10: //publish all and receive data
		//start publish
		runPublishWorker := TRUE;
		step := 20;
	20: IF HighSendPublish.finished THEN
		//wait until send is done		
			runPublishWorker := FALSE;
			step:= 30;

		END_IF
	30: //now check payload
		
			noData := FALSE;
		FOR i := 0 TO Count - 1 DO
			IF ReceivePayloadStore[i] <> SendPayloadStore[i] THEN
				noData := TRUE;
				EXIT;
			END_IF
		END_FOR
		IF NOT noData THEN
			step := 40;
			//unsubscripe
			subscribe := FALSE; 
		END_IF	
	40: 
		IF nextRun OR tNewRun.Q THEN 
			nextRun := FALSE;
			step := 0;
		END_IF
END_CASE

tNewRun(in := step = 40,PT:= repeatTime);

END_FUNCTION_BLOCK

// MQTT/TestCases/testHighLoadPublish
FUNCTION_BLOCK testHighLoadPublish
VAR_INPUT
	topics:UINT:=TEST_TOPICS;
	broker:STRING:='test.mosquitto.org:1883';
	addTopic:STRING(200);
	retpeatTime:TIME:=T#1M;
END_VAR
VAR_OUTPUT
END_VAR
VAR

	HighLoad:HighLoadPublish;

	init: BOOL;
	i:UINT;
	//testTopics:ARRAY[0..TOPICS_MAX] OF STRING(255);
	testTopic:STRING(255):='High Payload Test with very very very very very very very very very very big topic/Outs';
	
	testPayload:ARRAY[0..TOPICS_MAX]OF STRING(255);
	splitChar:STRING := '=';
	PayloadPrefix:STRING := 'Output:';
	
	
	ReceivePayloadStore:ARRAY[0..TOPICS_MAX] OF LINT;
	SendPayloadStore:ARRAY[0..TOPICS_MAX] OF STRING(255);
	SendPayloadStorePointerArray:ARRAY[0..TOPICS_MAX] OF POINTER TO STRING;
	tmpString:STRING;
	tmpString2:STRING;
	step:INT;
	nextRun: BOOL;
	tNewRun:ton;
	work:BOOL;


END_VAR
VAR CONSTANT
	TEST_TOPICS:UINT:= 200;
	TOPICS_MAX:UINT:=10000;
END_VAR

IF NOT init THEN
	 init := TRUE;
	//Testtopic();
	FOR i := 0 TO topics - 1 DO
		
		tmpString := PayloadPrefix;
		tmpString2 := UINT_TO_STRING(i);
		CommonTypesAndFunctions.concat(s1:= ADR(tmpString), s2:= ADR(tmpString2));
		
		CommonTypesAndFunctions.concat(s1:= ADR(tmpString), s2:= ADR(splitChar));
		CommonTypesAndFunctions.concat(s1:= ADR(tmpString), s2:= ADR(tmpString2));
		SendPayloadStore[i] := tmpString;
		SendPayloadStorePointerArray[i] := ADR(SendPayloadStore[i]);
		step := 10;
	END_FOR
	
END_IF

HighLoad(
	ClientID:= 'Test for HighLoadPublish', 
	Topic:= ADR(testTopic), 
	TopicFix:= TRUE, 
	payload:= ADR(SendPayloadStorePointerArray[0]),
	PayloadFix := FALSE, 
	CountArray:= topics, 
	UsedPublishFbs:= MyConstants.IN_OUT_SLOTS_SIZE - 1, 
	working:= work, 
	broker:= 'windows-10-pro:1883', 
	QoS:= QoS.ExactlyOnce, 
	RetainIn:= FALSE);

IF topics >= TOPICS_MAX THEN
	topics := TOPICS_MAX - 1;
END_IF


	
CASE step OF
	10: //empty
		step := 20;
	
	20: 
		work := TRUE; 
		step := 30;
	30: //wait for finish
		IF HighLoad.finished THEN
			work := FALSE;
			step := 40;
			
		END_IF
		
	40: //wait for next run
		IF tNewRun.Q OR nextRun THEN
			step := 10;
		END_IF 
END_CASE

tNewRun(in := step = 40,PT:= retpeatTime);

END_FUNCTION_BLOCK

// MQTT/Function Blocks/CallbackFBs/Callback Collector/CallbackCollector
(*this FB collects instances of FB with the MQTT_SUBSCRIBE_CALLBACK interface.
then you can pass a instance of this FB to a subscription FB to call all of your FBs to a specific subscription topic,
in this call you can check if the packet was for your instance. If your instance methode call return true, the the FB exits the
loop an so you may save cycle time.
MEmory for instance references are created dynamic, so no restriction by library*)
FUNCTION_BLOCK CallbackCollector IMPLEMENTS MQTT_SUBSCRIBE_CALLBACK
VAR_INPUT
END_VAR
VAR_OUTPUT
END_VAR
VAR
	first:POINTER TO CALLBACK_INSTANCES := 0;
	items:UDINT;
	size:UDINT;
END_VAR

//true if all ok, else false
METHOD put : BOOL
VAR_INPUT
	instance:MQTT_SUBSCRIBE_CALLBACK;
END_VAR
VAR
	aktElement:POINTER TO CALLBACK_INSTANCES;
END_VAR
aktElement := first;

IF aktElement = 0 THEN
	//first hit...
	{info 'semaphore'}
	first := __NEW(CALLBACK_INSTANCES);
	IF first = 0 THEN
		put := FALSE;
		RETURN;
	END_IF
	aktElement := first;
ELSE
	//search last
	WHILE aktElement^.next  <> 0 DO 
		aktElement := aktElement^.next; 
	END_WHILE
	{info 'semaphore'}
	aktElement^.next := __NEW(CALLBACK_INSTANCES);
	IF aktElement^.next = 0 THEN
		put := FALSE;
		RETURN;
	END_IF
	aktElement := aktElement^.next;
END_IF

aktElement^.callback := instance;
put := TRUE;
items := items + 1;
size := size + SIZEOF(CALLBACK_INSTANCES);
END_METHOD


METHOD PublishReceived : BOOL
VAR_INPUT
	(*Collection of received Data*)
	Data	: CALLBACK_DATA;
END_VAR
VAR
	element:POINTER TO CALLBACK_INSTANCES;
	loop: BOOL := true;

END_VAR


IF first = 0 THEN
	//no callback avalable
	RETURN;
END_IF
element := first;


WHILE loop DO
	IF element^.callback.PublishReceived(Data := Data) THEN
		PublishReceived := TRUE;
		RETURN;
	END_IF
	IF element^.next = 0 THEN
		loop := FALSE;
	ELSE
		element := element^.next;
	END_IF
END_WHILE
END_METHOD

//destroy all dynamic content
METHOD destroy : BOOL
VAR_INPUT
END_VAR
VAR
	aktElement:POINTER TO CALLBACK_INSTANCES;
	nextElement:POINTER TO CALLBACK_INSTANCES;
	


END_VAR
GVL_MQTT.ProgNum := PROG_NUM.DESTROY_CALLBACK_COLLECTOR;
IF first = 0 THEN
	RETURN;
END_IF

aktElement := first;

REPEAT
	nextElement := aktElement^.next;
	__DELETE(aktElement);
	aktElement := nextElement;
	items := items - 1;
	size := size - SIZEOF(CALLBACK_INSTANCES);
UNTIL aktElement = 0
END_REPEAT
first := 0;
GVL_MQTT.ProgNum := PROG_NUM.DESTROY_CALLBACK_COLLECTOR_DONE;
END_METHOD

METHOD FB_Exit : BOOL 
VAR_INPUT 
 bInCopyCode : BOOL; // TRUE: the exit method is called in order to leave the instance which will be copied afterwards (online change). 
END_VAR
destroy();
END_METHOD

END_FUNCTION_BLOCK

// MQTT/TestCases/Test Interfaces/FooBarReceivingFB
{attribute 'reflection'}
FUNCTION_BLOCK FooBarReceivingFB IMPLEMENTS MQTT_SUBSCRIBE_CALLBACK
VAR_INPUT
END_VAR
VAR_OUTPUT
END_VAR
VAR
	{attribute 'instance-path'}
	{attribute 'noinit'}
	instanceName: STRING(255);//this string contains the instance name of the FB
	//here we get the "lowest" element of the name...
	LastTreeName:STRING;
	//if set to true we search the instance name in the lowest topic
	splitTopic: BOOL;
	//if set to true we search the instance name in Payload separatet by the split char 
	splitPayload: BOOL;
	//an this is the split char...
	SplitPayloadChar: BYTE;
	(*here is the target where we will place the payload contend
	this can be anything...*)
	Target:STRING(255);
END_VAR

METHOD PublishReceived : BOOL
VAR_INPUT
	(*Collection of received Data*)
	Data	: CALLBACK_DATA;
	
END_VAR
VAR
	StrPt : POINTER TO STRING(255);
END_VAR
// no we can check if the topic/payload fits to my instance name.... 

//now search the right topic 
IF splitTopic THEN
	
	IF CommonTypesAndFunctions.StrEquals(str1:= Data.TopicOutSplit^.Topics[Data.TopicOutSplit^.ValidFields - 1], str2:= ADR(LastTreeName)) THEN
		Target := Data.PayloadString^;
	END_IF

END_IF

//now look into the payload
IF splitPayload THEN
	
